# B&R Automation Studio project Panasonic_LinkaPowerCP2_A2021055 (part 29)

#### Main.st - Init, cyclic, exit code
```iecst
PROGRAM _INIT
	(* Insert code here *)

END_PROGRAM

PROGRAM _CYCLIC

		//Volanie funkcie SequenceControl//
	SequenceControl(SC:= SC_P3_LeakageTestB);

	//Volanie podprogramov//
	OvlCentrovacky;
	OvlHornehoPritlaku;
	IOLinkKomunikacia;
	COM_Tester;

	//Reset sekcie //
	IF P3_LeakageTestB.Reset THEN
		SC_P3_LeakageTestB.Step:= 0;
		P3_LeakageTestB.Reset:= FALSE;
	ELSIF NOT Safety.STAV.Linka_ZonaCS_AKTIVNA THEN
		SC_P3_LeakageTestB.Step:= 0;
	END_IF

	CASE SC_P3_LeakageTestB.Step OF

		0:
			SC_P3_LeakageTestB.StepName:='0 - Nulovanie';
			SC_OvlCentrovacky.Step:= 0;
			SC_OvlHornehoPritlaku.Step:= 0;
			P3_LeakageTestB.Automat:= FALSE;
			P3_LeakageTestB.KoniecCyklu:= FALSE;
			P3_LeakageTestB.Manual:= FALSE;
			P3_LeakageTestB.STAV.PoINIT:= FALSE;
			P3_LeakageTestB.OUT.ZasunStoper:= FALSE;
			P3_LeakageTestB.OUT.Kopito_VYSUN:= FALSE;
			P3_LeakageTestB.OUT.Kopito_ZASUN:= TRUE;
			P3_LeakageTestB.RFID_hlava.PrecitajChipRFID:= FALSE;
			P3_LeakageTestB.CMD.RR_TestovaciaSekvencia_START:= FALSE;
			P3_LeakageTestB.CMD.RR_VysunSpodneKopito:= FALSE;
			P3_LeakageTestB.CMD.RR_HornyPritlak_VYSUN:= FALSE;
			P3_LeakageTestB.CMD.RR_HornyPritlak_ZASUN:= FALSE;
			P3_LeakageTestB.STAV.RR_TestovaciaSekvencia_BUSY:= FALSE;
			TRCB_P3_LeakageTestB_ST8B.CMD.VyziadajStavPaletky_TYP1:= FALSE;
			TRCB_P3_LeakageTestB_ST8B.CMD.PriradQRkodFiltra_TYP3:= FALSE;
			TRCB_P3_LeakageTestB_ST8B.CMD.OdosliStavPaletky_TYP2:= FALSE;
			TRCB_P3_LeakageTestB_ST8B.CMD.VyziadajStavPanatrace_TYP4:= FALSE;
			AteqLeakageTester_B.CitajParametreTestera:= FALSE;
			AteqLeakageTester_B.START_Testovania:= FALSE;
			P34_Vizu.ZobrazHL2_ST8:= FALSE;
			P34_Vizu.ZobrazHL4_ST8:= FALSE;
			TRCB_P3_LeakTestB_OpatovnyDopyt:= FALSE;
			TRCB_P3_LeakTestB_PaletkaNG:= FALSE;
			PocetDopytovNaServer:= 0;
			PocetOpakovaniTestu:= 0;
			OpakovanyTest:= FALSE;
			TestovaciKus:= FALSE;
			P3_LeakageTestB_Taktime.IN.START_MeraniaCasu:= FALSE;
			P3_LeakageTestB_Taktime.IN.START_MeraniaStratovehoCasu:= FALSE;

			P3_ZdvizkaPredLeakTestB.STAV.PrebiehaVyvezeniePaletky:= FALSE;
			P3_LeakageTestB.STAV.PrebiehaVyvezeniePaletky:= FALSE;

			IF Safety.STAV.Linka_ZonaCS_AKTIVNA AND
				Safety.STAV.P3_ZonaBunky_AKTIVNA AND
				P3_Pracovisko.STAV.HardwareBunky_OK AND
				NOT P3_Pracovisko.STAV.Porucha_ST1 AND
				NOT P3_Pracovisko.STAV.Porucha_ST2 AND
				NOT P3_Pracovisko.STAV.Porucha_ST3 AND
				NOT P3_Pracovisko.STAV.Porucha_ST4 AND
				NOT P3_Pracovisko.STAV.Porucha_ST5 AND
				NOT P3_Pracovisko.STAV.Porucha_ST6 AND
				NOT P3_Pracovisko.STAV.Porucha_ST7 AND
				NOT P3_Pracovisko.STAV.Porucha_ST8 THEN
				SC_P3_LeakageTestB.ResetStep:= TRUE;
				SC_P3_LeakageTestB.Step:= 1;
			END_IF

		1:
			SC_P3_LeakageTestB.StepName:='1 - Cakam na spustenie vyroby';
			P3_LeakageTestB.KoniecCyklu:= FALSE;
			IF P3_LeakageTestB.Automat THEN
				SC_P3_LeakageTestB.Step:= 2;
			ELSIF P3_LeakageTestB.Manual THEN
				SC_P3_LeakageTestB.Step:= 700;
			END_IF

			//********************************************************Inicializácia****************************************************************************//

		2:
			SC_P3_LeakageTestB.StepName:='2 - Inicializacia - cakam na spustenie inicializacie';
			SC_P3_LeakageTestB.IdleTime.PT:= T#500ms;
			SC_P3_LeakageTestB.AlarmTime.PT:= T#5s;
			SC_P3_LeakageTestB.IdleTime.IN:= TRUE;

			IF SC_P3_LeakageTestB.IdleTime.Q THEN
				SC_P3_LeakageTestB.ResetStep:= TRUE;
				SC_P3_LeakageTestB.Step:= 5;
			END_IF

		5:
			SC_P3_LeakageTestB.StepName:='5 - Inicializacia - zasunutie horneho pritlaku';
			SC_P3_LeakageTestB.IdleTime.PT:= T#2s;
			SC_P3_LeakageTestB.AlarmTime.PT:= T#5s;

			IF NOT SC_P3_LeakageTestB.Switch1 THEN
				HornyPritlak_ZASUN:= TRUE;
				SC_P3_LeakageTestB.Switch1:= TRUE;
			END_IF

			IF P3_LeakageTestB.IN.HornyPritlak_ZASUNUTY THEN
				SC_P3_LeakageTestB.ResetStep:= TRUE;
				SC_P3_LeakageTestB.Step:= 8;
			END_IF

		8:
			SC_P3_LeakageTestB.StepName:='8 - Inicializacia - zasunutie centrovacky';
			SC_P3_LeakageTestB.IdleTime.PT:= T#4s;
			SC_P3_LeakageTestB.AlarmTime.PT:= T#5s;

			IF NOT SC_P3_LeakageTestB.Switch1 THEN
				Centrovacku_ZASUN:= TRUE;
				SC_P3_LeakageTestB.Switch1:= TRUE;
			END_IF

			IF P3_LeakageTestB.IN.Centrovanie_ZASUNUTE THEN
				SC_P3_LeakageTestB.ResetStep:= TRUE;
				SC_P3_LeakageTestB.Step:= 10;
			END_IF

		10:
			SC_P3_LeakageTestB.StepName:='10 - Inicializacia - kontrola typu zalozeneho kopita';
			SC_P3_LeakageTestB.IdleTime.PT:= T#4s;
			SC_P3_LeakageTestB.AlarmTime.PT:= T#5s;

			IF Linka.PAR.ZvolenyModel = '4F' AND P3_LeakageTestB.IN.PritomnostKopita AND P3_LeakageTestB.IN.Tester_TypKonektoru_4F THEN
				SC_P3_LeakageTestB.ResetStep:= TRUE;
				SC_P3_LeakageTestB.Step:= 13;
			ELSIF Linka.PAR.ZvolenyModel = '5F' AND P3_LeakageTestB.IN.PritomnostKopita AND P3_LeakageTestB.IN.Tester_TypKonektoru_5F_5H THEN
				SC_P3_LeakageTestB.ResetStep:= TRUE;
				SC_P3_LeakageTestB.Step:= 13;
			ELSIF Linka.PAR.ZvolenyModel = '5H' AND P3_LeakageTestB.IN.PritomnostKopita AND P3_LeakageTestB.IN.Tester_TypKonektoru_5F_5H THEN
				SC_P3_LeakageTestB.ResetStep:= TRUE;
				SC_P3_LeakageTestB.Step:= 13;
			ELSE
				P34_Alarmy[315]:= TRUE;
				P3_Pracovisko.STAV.Porucha_ST6:= TRUE;
			END_IF

		13:
			SC_P3_LeakageTestB.StepName:='13 - Inicializacia - hladanie paletky';
			SC_P3_LeakageTestB.IdleTime.PT:= T#5s;
			SC_P3_LeakageTestB.AlarmTime.PT:= T#5s;

			SC_P3_LeakageTestB.IdleTime.IN:= P3_Dopravniky.STAV.PoINIT;

			IF P3_LeakageTestB.CMD.RR_TestovaciaSekvencia_START THEN
				SC_P3_LeakageTestB.ResetStep:= TRUE;
				SC_P3_LeakageTestB.Step:= 120;
			ELSIF P3_LeakageTestB.RFID_hlava.PritomnostPaletky THEN
				SC_P3_LeakageTestB.ResetStep:= TRUE;
				SC_P3_LeakageTestB.Step:= 20;
			ELSIF SC_P3_LeakageTestB.IdleTime.Q THEN
				P3_LeakageTestB.STAV.PoINIT:= TRUE;
				SC_P3_LeakageTestB.ResetStep:= TRUE;
				SC_P3_LeakageTestB.Step:= 100;
			END_IF

		20:
			SC_P3_LeakageTestB.StepName:='20 - Inicializacia - precitanie cisla paletky';
			SC_P3_LeakageTestB.IdleTime.PT:= T#200ms;
			SC_P3_LeakageTestB.AlarmTime.PT:= T#5s;

			SC_P3_LeakageTestB.IdleTime.IN:= P3_LeakageTestB.RFID_hlava.PritomnostPaletky;

			IF SC_P3_LeakageTestB.IdleTime.Q AND NOT SC_P3_LeakageTestB.Switch1 THEN
				P3_LeakageTestB.RFID_hlava.PrecitajChipRFID:= TRUE;
				i:= 0;
				SC_P3_LeakageTestB.Switch1:= TRUE;
			END_IF

			IF P3_LeakageTestB.RFID_hlava.Stav_CitanieZapis_OK AND P3_LeakageTestB.RFID_hlava.PrecitaneCisloPaletky <> 0 THEN
				i:= P3_LeakageTestB.RFID_hlava.PrecitaneCisloPaletky;
				P3_LeakageTestB.PAR.CisloPaletky:= P3_LeakageTestB.RFID_hlava.PrecitaneCisloPaletky;
				P3_LeakageTestB.RFID_hlava.PrecitajChipRFID:= FALSE;
				SC_P3_LeakageTestB.ResetStep:= TRUE;
				SC_P3_LeakageTestB.Step:= 23;
			END_IF

		23:
			SC_P3_LeakageTestB.StepName:='23 - Inicializacia - priradenie indexu paletky na zaklade precitanej hodnoty';
			SC_P3_LeakageTestB.IdleTime.PT:= T#200ms;
			SC_P3_LeakageTestB.AlarmTime.PT:= T#5s;

			IF i<> 0 THEN
				P3_LeakageTestB.PAR.CisloPaletky_STRING:= USINT_TO_STRING(i);
				Paletka[i].PAR.CisloPaletky:= USINT_TO_STRING(i);
				SC_P3_LeakageTestB.ResetStep:= TRUE;
				SC_P3_LeakageTestB.Step:= 30;
			ELSE
				P34_Alarmy[312]:= TRUE;
				P3_Pracovisko.STAV.Porucha_ST6:= TRUE;
			END_IF

		30:
			SC_P3_LeakageTestB.StepName:='30 - Inicializacia - kontrola stavu paletky';
			SC_P3_LeakageTestB.IdleTime.PT:= T#200ms;
			SC_P3_LeakageTestB.AlarmTime.PT:= T#5s;

			IF Paletka[i].STAV.StavPaletky = '' THEN
				Paletka[i].STAV.StavPaletky:= 'NG';
				SC_P3_LeakageTestB.ResetStep:= TRUE;
				SC_P3_LeakageTestB.Step:= 560;
			ELSIF Paletka[i].STAV.StavPaletky = 'PRECH' THEN
				P3_LeakageTestB.STAV.PoINIT:= TRUE;
				SC_P3_LeakageTestB.ResetStep:= TRUE;
				SC_P3_LeakageTestB.Step:= 560;
			ELSIF Paletka[i].STAV.StavPaletky = 'TEST' AND Paletka[i].STAV.CisloTestovacejStanice = 'ST_8A,8B' THEN
				IF P3_LeakageTestB.STAV.Tester_ON THEN
					TestovaciKus:= TRUE;
					P3_LeakageTestB.STAV.PoINIT:= TRUE;
					SC_P3_LeakageTestB.ResetStep:= TRUE;
					SC_P3_LeakageTestB.Step:= 110;
				ELSE
					P3_LeakageTestB.STAV.PoINIT:= TRUE;
					SC_P3_LeakageTestB.ResetStep:= TRUE;
					SC_P3_LeakageTestB.Step:= 560;
				END_IF
			ELSIF Paletka[i].STAV.StavPaletky = 'TEST' AND Paletka[i].STAV.CisloTestovacejStanice <> 'ST_8A,8B' THEN
				P3_LeakageTestB.STAV.PoINIT:= TRUE;
				SC_P3_LeakageTestB.ResetStep:= TRUE;
				SC_P3_LeakageTestB.Step:= 560;
			ELSIF Paletka[i].STAV.StavPaletky = 'REV' AND Paletka[i].STAV.CisloRevorkovejStanice = 'ST_8A,8B' THEN
				IF P3_LeakageTestB.STAV.Tester_ON THEN
					Paletka[i].STAV.StavPaletky:= 'OK';
					P3_LeakageTestB.STAV.PoINIT:= TRUE;
					SC_P3_LeakageTestB.ResetStep:= TRUE;
					SC_P3_LeakageTestB.Step:= 110;
				ELSE
					P3_LeakageTestB.STAV.PoINIT:= TRUE;
					SC_P3_LeakageTestB.ResetStep:= TRUE;
					SC_P3_LeakageTestB.Step:= 560;
				END_IF
			ELSIF Paletka[i].STAV.StavPaletky = 'REV' AND Paletka[i].STAV.CisloRevorkovejStanice <> 'ST_8A,8B' THEN
				P3_LeakageTestB.STAV.PoINIT:= TRUE;
				SC_P3_LeakageTestB.ResetStep:= TRUE;
				SC_P3_LeakageTestB.Step:= 560;
			ELSIF Paletka[i].STAV.StavPaletky = 'OK' THEN
				IF P3_LeakageTestB.STAV.Tester_ON THEN
					SC_P3_LeakageTestB.ResetStep:= TRUE;
					SC_P3_LeakageTestB.Step:= 33;
				ELSE
					P3_LeakageTestB.STAV.PoINIT:= TRUE;
					SC_P3_LeakageTestB.ResetStep:= TRUE;
					SC_P3_LeakageTestB.Step:= 560;
				END_IF
			ELSIF Paletka[i].STAV.StavPaletky = 'NG' THEN
				P3_LeakageTestB.STAV.PoINIT:= TRUE;
				SC_P3_LeakageTestB.ResetStep:= TRUE;
				SC_P3_LeakageTestB.Step:= 560;
			END_IF

		33:
			SC_P3_LeakageTestB.StepName:='33 - Inicializacia - kontrola uzavretia komunikacie';
			SC_P3_LeakageTestB.IdleTime.PT:= T#200ms;
			SC_P3_LeakageTestB.AlarmTime.PT:= T#5s;

			IF Paletka[i].STAV.Komunikacia_DONE THEN
				P3_LeakageTestB.STAV.PoINIT:= TRUE;
				SC_P3_LeakageTestB.ResetStep:= TRUE;
				SC_P3_LeakageTestB.Step:= 560;
			ELSE
				P3_LeakageTestB.STAV.PoINIT:= TRUE;
				SC_P3_LeakageTestB.ResetStep:= TRUE;
				SC_P3_LeakageTestB.Step:= 100;
			END_IF

			//********************************************************Automatický režim****************************************************************************//

		100:
			SC_P3_LeakageTestB.StepName:='100 - Automaticky Rezim - cakam na príchod paletky na stoper';
			SC_P3_LeakageTestB.IdleTime.PT:= T#200ms;
			SC_P3_LeakageTestB.AlarmTime.PT:= T#5s;

			SC_P3_LeakageTestB.IdleTime.IN:= P3_LeakageTestB.RFID_hlava.PritomnostPaletky;

			IF P3_LeakageTestB.RFID_hlava.PritomnostPaletky THEN
				P3_ZdvizkaPredLeakTestB.STAV.PrebiehaVyvezeniePaletky:= FALSE;
			END_IF

			IF NOT SC_P3_LeakageTestB.Switch1 AND P3_LeakageTestB.RFID_hlava.PritomnostPaletky THEN
				P3_LeakageTestB_Taktime.IN.START_MeraniaCasu:= TRUE;
				P3_LeakageTestB_Taktime.IN.ZAPIS_MeraniaCasu:= TRUE;
				P3_LeakageTestB_Taktime.IN.ZAPIS_StratovyCas:= TRUE;
				Buffer_10.Hodnota:= P3_LeakageTestB_Taktime.OUT.StratoveSekundy;
				Buffer_10.ZapisHodnotu:= TRUE;
				SC_P3_LeakageTestB.Switch1:= TRUE;
			END_IF

			IF P3_LeakageTestB.KoniecCyklu THEN
				SC_P3_LeakageTestB.ResetStep:= TRUE;
				SC_P3_LeakageTestB.Step:= 0;
			ELSIF SC_P3_LeakageTestB.IdleTime.Q THEN
				SC_P3_LeakageTestB.ResetStep:= TRUE;
				SC_P3_LeakageTestB.Step:= 101;
			END_IF

		101:
			SC_P3_LeakageTestB.StepName:='101 - Automaticky Rezim - precitanie cisla paletky';
			SC_P3_LeakageTestB.IdleTime.PT:= T#200ms;
			SC_P3_LeakageTestB.AlarmTime.PT:= T#5s;
			SC_P3_LeakageTestB.IdleTime.IN:= TRUE;

			IF NOT SC_P3_LeakageTestB.Switch1 THEN
				P3_LeakageTestB.RFID_hlava.PrecitajChipRFID:= TRUE;
				i:= 0;
				SC_P3_LeakageTestB.Switch1:= TRUE;
			END_IF

			IF P3_LeakageTestB.RFID_hlava.Stav_CitanieZapis_OK AND P3_LeakageTestB.RFID_hlava.PrecitaneCisloPaletky <> 0 THEN
				i:= P3_LeakageTestB.RFID_hlava.PrecitaneCisloPaletky;
				P3_LeakageTestB.PAR.CisloPaletky:= P3_LeakageTestB.RFID_hlava.PrecitaneCisloPaletky;
				P3_LeakageTestB.RFID_hlava.PrecitajChipRFID:= FALSE;
				SC_P3_LeakageTestB.ResetStep:= TRUE;
				SC_P3_LeakageTestB.Step:= 102;
			END_IF

		102:
			SC_P3_LeakageTestB.StepName:='102 - Automaticky Rezim - priradenie indexu paletky na zaklade precitanej hodnoty';
			SC_P3_LeakageTestB.IdleTime.PT:= T#200ms;
			SC_P3_LeakageTestB.AlarmTime.PT:= T#5s;

			IF i<> 0 THEN
				P3_LeakageTestB.PAR.CisloPaletky_STRING:= USINT_TO_STRING(i);
				Paletka[i].PAR.CisloPaletky:= USINT_TO_STRING(i);
				SC_P3_LeakageTestB.ResetStep:= TRUE;
				SC_P3_LeakageTestB.Step:= 103;
			ELSE
				P34_Alarmy[312]:= TRUE;
				P3_Pracovisko.STAV.Porucha_ST6:= TRUE;
			END_IF

		103:
			SC_P3_LeakageTestB.StepName:='103 - Automaticky Rezim - kontrola stavu paletky';
			SC_P3_LeakageTestB.IdleTime.PT:= T#200ms;
			SC_P3_LeakageTestB.AlarmTime.PT:= T#5s;

			IF Paletka[i].STAV.StavPaletky = '' THEN
				Paletka[i].STAV.StavPaletky:= 'NG';
				SC_P3_LeakageTestB.ResetStep:= TRUE;
				SC_P3_LeakageTestB.Step:= 560;
			ELSIF Paletka[i].STAV.StavPaletky = 'PRECH' THEN
				SC_P3_LeakageTestB.ResetStep:= TRUE;
				SC_P3_LeakageTestB.Step:= 560;
			ELSIF Paletka[i].STAV.StavPaletky = 'TEST' AND Paletka[i].STAV.CisloTestovacejStanice = 'ST_8A,8B' THEN
				IF P3_LeakageTestB.STAV.Tester_ON THEN
					TestovaciKus:= TRUE;
					SC_P3_LeakageTestB.ResetStep:= TRUE;
					SC_P3_LeakageTestB.Step:= 110;
				ELSE
					SC_P3_LeakageTestB.ResetStep:= TRUE;
					SC_P3_LeakageTestB.Step:= 560;
				END_IF
			ELSIF Paletka[i].STAV.StavPaletky = 'TEST' AND Paletka[i].STAV.CisloTestovacejStanice <> 'ST_8A,8B' THEN
				SC_P3_LeakageTestB.ResetStep:= TRUE;
				SC_P3_LeakageTestB.Step:= 560;
			ELSIF Paletka[i].STAV.StavPaletky = 'REV' AND Paletka[i].STAV.CisloRevorkovejStanice = 'ST_8A,8B' THEN
				IF P3_LeakageTestB.STAV.Tester_ON THEN
					Paletka[i].STAV.StavPaletky:= 'OK';
					SC_P3_LeakageTestB.ResetStep:= TRUE;
					SC_P3_LeakageTestB.Step:= 110;
				ELSE
					SC_P3_LeakageTestB.ResetStep:= TRUE;
					SC_P3_LeakageTestB.Step:= 560;
				END_IF
			ELSIF Paletka[i].STAV.StavPaletky = 'REV' AND Paletka[i].STAV.CisloRevorkovejStanice <> 'ST_8A,8B' THEN
				SC_P3_LeakageTestB.ResetStep:= TRUE;
				SC_P3_LeakageTestB.Step:= 560;
			ELSIF Paletka[i].STAV.StavPaletky = 'OK' THEN
				IF P3_LeakageTestB.STAV.Tester_ON THEN
					SC_P3_LeakageTestB.ResetStep:= TRUE;
					SC_P3_LeakageTestB.Step:= 110;
				ELSE
					SC_P3_LeakageTestB.ResetStep:= TRUE;
					SC_P3_LeakageTestB.Step:= 560;
				END_IF
			ELSIF Paletka[i].STAV.StavPaletky = 'NG' THEN
				SC_P3_LeakageTestB.ResetStep:= TRUE;
				SC_P3_LeakageTestB.Step:= 560;
			END_IF

		110:
			SC_P3_LeakageTestB.StepName:='110 - Automaticky Rezim - vyziadanie stavu komunikacie zo serverom';
			SC_P3_LeakageTestB.IdleTime.PT:= T#200ms;
			SC_P3_LeakageTestB.AlarmTime.PT:= T#10s;

			IF Linka.KOM_Panatrace_OFF THEN
				SC_P3_LeakageTestB.ResetStep:= TRUE;
				SC_P3_LeakageTestB.Step:= 120;
			ELSIF NOT SC_P3_LeakageTestB.Switch1 THEN
				TRCB_P3_LeakageTestB_ST8B.CMD.VyziadajStavPanatrace_TYP4:= TRUE;
				Centrovacku_VYSUN:= TRUE;
				P3_LeakageTestB_Taktime.IN.START_MeraniaStratovehoCasu:= TRUE;
				SC_P3_LeakageTestB.Switch1:= TRUE;
			END_IF

			IF TRCB_P3_LeakageTestB_ST8B.STATUS.KomunikaciaUkoncena THEN
				TRCB_P3_LeakageTestB_ST8B.CMD.VyziadajStavPanatrace_TYP4:= FALSE;
				P3_LeakageTestB_Taktime.IN.START_MeraniaStratovehoCasu:= FALSE;
				SC_P3_LeakageTestB.ResetStep:= TRUE;
				SC_P3_LeakageTestB.Step:= 111;
			ELSIF TRCB_P3_LeakageTestB_ST8B.STATUS.KomunikaciaError THEN
				TRCB_P3_LeakageTestB_ST8B.CMD.VyziadajStavPanatrace_TYP4:= FALSE;
				P3_LeakageTestB_Taktime.IN.START_MeraniaStratovehoCasu:= FALSE;
				SC_P3_LeakageTestB.ResetStep:= TRUE;
				SC_P3_LeakageTestB.Step:= 112;
			END_IF

		111:
			SC_P3_LeakageTestB.StepName:='111 - Automaticky Rezim - kontrola odpovede servera';
			SC_P3_LeakageTestB.IdleTime.PT:= T#200ms;
			SC_P3_LeakageTestB.AlarmTime.PT:= T#5s;

			IF NOT TRCB_P3_LeakageTestB_ST8B.STATUS.KomunikaciaUkoncena THEN
				IF TRCB_P3_LeakageTestB_ST8B.OUTPUTS.DruhCinnostiNaPaletke = '0;Generating' THEN
					SC_P3_LeakageTestB.ResetStep:= TRUE;
					SC_P3_LeakageTestB.Step:= 112;
				ELSIF TRCB_P3_LeakageTestB_ST8B.OUTPUTS.DruhCinnostiNaPaletke = '1;Request' THEN
					SC_P3_LeakageTestB.ResetStep:= TRUE;
					SC_P3_LeakageTestB.Step:= 115;
				ELSIF TRCB_P3_LeakageTestB_ST8B.OUTPUTS.DruhCinnostiNaPaletke = '2;Report' THEN
					SC_P3_LeakageTestB.ResetStep:= TRUE;
					SC_P3_LeakageTestB.Step:= 120;
				ELSIF TRCB_P3_LeakageTestB_ST8B.OUTPUTS.DruhCinnostiNaPaletke = '3;Wedding' THEN
					SC_P3_LeakageTestB.ResetStep:= TRUE;
					SC_P3_LeakageTestB.Step:= 112;
				ELSIF TRCB_P3_LeakageTestB_ST8B.OUTPUTS.DruhCinnostiNaPaletke = '4;Status' THEN
					SC_P3_LeakageTestB.ResetStep:= TRUE;
					SC_P3_LeakageTestB.Step:= 112;
				ELSIF TRCB_P3_LeakageTestB_ST8B.OUTPUTS.DruhCinnostiNaPaletke = '5;' THEN
					SC_P3_LeakageTestB.ResetStep:= TRUE;
					SC_P3_LeakageTestB.Step:= 112;
				ELSE
					SC_P3_LeakageTestB.ResetStep:= TRUE;
					SC_P3_LeakageTestB.Step:= 112;
				END_IF
			END_IF

		112:
			SC_P3_LeakageTestB.StepName:='112 - Automaticky Rezim - rozhodnutie obsluhy po chybe komunikacie s Panatrace';
			SC_P3_LeakageTestB.IdleTime.PT:= T#200ms;
			SC_P3_LeakageTestB.AlarmTime.PT:= T#5s;

			P34_Vizu.ZobrazHL4_ST8:= TRUE;

			IF TRCB_P3_LeakTestB_OpatovnyDopyt THEN
				TRCB_P3_LeakTestB_OpatovnyDopyt:= FALSE;
				P34_Vizu.ZobrazHL4_ST8:= FALSE;
				SC_P3_LeakageTestB.ResetStep:= TRUE;
				SC_P3_LeakageTestB.Step:= 110;
			ELSIF TRCB_P3_LeakTestB_PaletkaNG THEN
				TRCB_P3_LeakTestB_PaletkaNG:= FALSE;
				P34_Vizu.ZobrazHL4_ST8:= FALSE;
				Paletka[i].STAV.StavPaletky := 'NG';
				SC_P3_LeakageTestB.ResetStep:= TRUE;
				SC_P3_LeakageTestB.Step:= 118;
			END_IF

		115:
			SC_P3_LeakageTestB.StepName:='115 - Automaticky Rezim - vyziadanie stavu paletky zo servera, zacentrovanie paletky';
			SC_P3_LeakageTestB.IdleTime.PT:= T#200ms;
			SC_P3_LeakageTestB.AlarmTime.PT:= T#5s;
			SC_P3_LeakageTestB.IdleTime.IN:= TRUE;

			IF NOT SC_P3_LeakageTestB.Switch1 AND TRCB_P3_LeakageTestB_ST8B.STATUS.KOM_READY THEN
				TRCB_P3_LeakageTestB_ST8B.CMD.VyziadajStavPaletky_TYP1:= TRUE;
				P3_LeakageTestB_Taktime.IN.START_MeraniaStratovehoCasu:= TRUE;
				SC_P3_LeakageTestB.Switch1:= TRUE;
			END_IF

			IF TRCB_P3_LeakageTestB_ST8B.STATUS.KomunikaciaUkoncena THEN
				TRCB_P3_LeakageTestB_ST8B.CMD.VyziadajStavPaletky_TYP1:= FALSE;
				P3_LeakageTestB_Taktime.IN.START_MeraniaStratovehoCasu:= FALSE;
				SC_P3_LeakageTestB.ResetStep:= TRUE;
				SC_P3_LeakageTestB.Step:= 116;
			ELSIF TRCB_P3_LeakageTestB_ST8B.STATUS.KomunikaciaError THEN
				TRCB_P3_LeakageTestB_ST8B.CMD.VyziadajStavPaletky_TYP1:= FALSE;
				P3_LeakageTestB_Taktime.IN.START_MeraniaStratovehoCasu:= FALSE;
				SC_P3_LeakageTestB.ResetStep:= TRUE;
				SC_P3_LeakageTestB.Step:= 112;
			END_IF

		116:
			SC_P3_LeakageTestB.StepName:='116 - Automaticky Rezim - kontrola odpovede servera';
			SC_P3_LeakageTestB.IdleTime.PT:= T#200ms;
			SC_P3_LeakageTestB.AlarmTime.PT:= T#5s;

			IF NOT TRCB_P3_LeakageTestB_ST8B.STATUS.KomunikaciaUkoncena AND P3_LeakageTestB.IN.Centrovanie_VYSUNUTE THEN
				IF TRCB_P3_LeakageTestB_ST8B.OUTPUTS.PovolenieCinnostiNaPaletke = 'OK' THEN
					IF TRCB_P3_LeakageTestB_ST8B.OUTPUTS.DruhCinnostiNaPaletke  = 'PRD;ST8B' THEN
						SC_P3_LeakageTestB.ResetStep:= TRUE;
						SC_P3_LeakageTestB.Step:= 120;
					ELSIF TRCB_P3_LeakageTestB_ST8B.OUTPUTS.DruhCinnostiNaPaletke  = 'SMP;ST8A,ST8B' THEN
						SC_P3_LeakageTestB.ResetStep:= TRUE;
						SC_P3_LeakageTestB.Step:= 120;
					ELSIF TRCB_P3_LeakageTestB_ST8B.OUTPUTS.DruhCinnostiNaPaletke  = 'PRD;ST8A,ST8B' THEN
						SC_P3_LeakageTestB.ResetStep:= TRUE;
						SC_P3_LeakageTestB.Step:= 120;
					END_IF
				ELSIF TRCB_P3_LeakageTestB_ST8B.OUTPUTS.PovolenieCinnostiNaPaletke = 'NG' THEN
					SC_P3_LeakageTestB.ResetStep:= TRUE;
					SC_P3_LeakageTestB.Step:= 117;
				END_IF
			END_IF

		117:
			SC_P3_LeakageTestB.StepName:='115 - Automaticky Rezim - rozhodnutie obsluhy po odpovedi panatrace NG';
			SC_P3_LeakageTestB.IdleTime.PT:= T#200ms;
			SC_P3_LeakageTestB.AlarmTime.PT:= T#5s;

			P34_Vizu.ZobrazHL2_ST8:= TRUE;

			IF TRCB_P3_LeakTestB_OpatovnyDopyt THEN
				TRCB_P3_LeakTestB_OpatovnyDopyt:= FALSE;
				P34_Vizu.ZobrazHL2_ST8:= FALSE;
				SC_P3_LeakageTestB.ResetStep:= TRUE;
				SC_P3_LeakageTestB.Step:= 110;
			ELSIF TRCB_P3_LeakTestB_PaletkaNG THEN
				TRCB_P3_LeakTestB_PaletkaNG:= FALSE;
				P34_Vizu.ZobrazHL2_ST8:= FALSE;
				Paletka[i].STAV.StavPaletky := 'NG';
				SC_P3_LeakageTestB.ResetStep:= TRUE;
				SC_P3_LeakageTestB.Step:= 118;
			END_IF

		118:
			SC_P3_LeakageTestB.StepName:='118 - Automaticky Rezim - odcentrovanie paletky po odpovedi servera NG';
			SC_P3_LeakageTestB.IdleTime.PT:= T#200ms;
			SC_P3_LeakageTestB.AlarmTime.PT:= T#5s;

			IF NOT SC_P3_LeakageTestB.Switch1 THEN
				Centrovacku_ZASUN:= TRUE;
				SC_P3_LeakageTestB.Switch1:= TRUE;
			END_IF

			IF P3_LeakageTestB.IN.Centrovanie_ZASUNUTE THEN
				SC_P3_LeakageTestB.ResetStep:= TRUE;
				SC_P3_LeakageTestB.Step:= 560;
			END_IF

			//Zatvorenie Leakage testera//

		120:
			SC_P3_LeakageTestB.StepName:='120 - Automaticky Rezim - zacentrovanie paletky ';
			SC_P3_LeakageTestB.IdleTime.PT:= T#200ms;
			SC_P3_LeakageTestB.AlarmTime.PT:= T#5s;

			IF NOT SC_P3_LeakageTestB.Switch1 THEN
				Centrovacku_VYSUN:= TRUE;
				SC_P3_LeakageTestB.Switch1:= TRUE;
			END_IF

			IF P3_LeakageTestB.IN.Centrovanie_VYSUNUTE THEN
				SC_P3_LeakageTestB.ResetStep:= TRUE;
				SC_P3_LeakageTestB.Step:= 123;
			END_IF

		123:
			SC_P3_LeakageTestB.StepName:='123 - Automaticky Rezim - vysunutie horneho pritlaku ';
			SC_P3_LeakageTestB.IdleTime.PT:= T#3s;
			SC_P3_LeakageTestB.AlarmTime.PT:= T#5s;

			IF NOT SC_P3_LeakageTestB.Switch1 THEN
				HornyPritlak_VYSUN:= TRUE;
				SC_P3_LeakageTestB.Switch1:= TRUE;
			END_IF

			IF P3_LeakageTestB.IN.HornyPritlak_VYSUNUTY THEN
				SC_P3_LeakageTestB.ResetStep:= TRUE;
				SC_P3_LeakageTestB.Step:= 125;
			END_IF

		125:
			SC_P3_LeakageTestB.StepName:='125 - Automaticky Rezim - vysunutie spodneho kopita';
			SC_P3_LeakageTestB.IdleTime.PT:= T#1s;
			SC_P3_LeakageTestB.AlarmTime.PT:= T#5s;
			SC_P3_LeakageTestB.IdleTime.IN:= TRUE;

			IF P3_LeakageTestB.IN.PritomnostKopita AND P3_LeakageTestB.IN.Kopito_ZASUNUTE THEN
				P3_LeakageTestB.OUT.Kopito_ZASUN:= FALSE;
				P3_LeakageTestB.OUT.Kopito_VYSUN:= TRUE;
				SC_P3_LeakageTestB.ResetStep:= TRUE;
				SC_P3_LeakageTestB.Step:= 128;
			END_IF

		128:
			SC_P3_LeakageTestB.StepName:='128 - Automaticky Rezim - cakam na vysunutie kopita';
			SC_P3_LeakageTestB.IdleTime.PT:= T#200ms;
			SC_P3_LeakageTestB.AlarmTime.PT:= T#300ms;

			SC_P3_LeakageTestB.IdleTime.IN:= NOT P3_LeakageTestB.IN.Kopito_ZASUNUTE;

			IF SC_P3_LeakageTestB.IdleTime.Q THEN
				P3_LeakageTestB.OUT.PneuZamokCentrovania_ODOMKNI:= FALSE;
				P3_LeakageTestB.OUT.PneuZamokZvonu_ODOMKNI:= FALSE;
				SC_P3_LeakageTestB.ResetStep:= TRUE;
				SC_P3_LeakageTestB.Step:= 130;
			END_IF

		130:
			SC_P3_LeakageTestB.StepName:='130 - Automaticky Rezim - spustenie testera';
			SC_P3_LeakageTestB.IdleTime.PT:= T#4s800ms;
			SC_P3_LeakageTestB.AlarmTime.PT:= T#5s;

			IF NOT SC_P3_LeakageTestB.Switch1 AND AteqLeakageTester_B.Stav_READY THEN
				AteqLeakageTester_B.START_Testovania:= TRUE;
				SC_P3_LeakageTestB.IdleTime.IN:= TRUE;
				SC_P3_LeakageTestB.Switch1:= TRUE;
			END_IF

			IF NOT AteqLeakageTester_B.Stav_READY AND AteqLeakageTester_B.Stav_START_DONE AND NOT AteqLeakageTester_B.VysledokTestovania_OK AND NOT AteqLeakageTester_B.VysledokTestovania_NG AND SC_P3_LeakageTestB.IdleTime.Q THEN
				SC_P3_LeakageTestB.ResetStep:= TRUE;
				SC_P3_LeakageTestB.Step:= 133;
			END_IF

		133:
			SC_P3_LeakageTestB.StepName:='133 - Automaticky Rezim - nacitanie parametrov testera';
			SC_P3_LeakageTestB.IdleTime.PT:= T#500ms;
			SC_P3_LeakageTestB.AlarmTime.PT:= T#5s;

			IF AteqLeakageTester_B.Stav_READY THEN
				AteqLeakageTester_B.START_Testovania:= FALSE;
				AteqLeakageTester_B.CitajParametreTestera:= TRUE;
			END_IF

			SC_P3_LeakageTestB.IdleTime.IN:= AteqLeakageTester_B.Stav_CitanieParametrov_OK;

			IF AteqLeakageTester_B.Stav_CitanieParametrov_OK AND SC_P3_LeakageTestB.IdleTime.Q THEN
				Reports.LeakageTest.CasPlnenia.StanicaB:= REAL_TO_STRING(AteqLeakageTester_B.CasPnenia);
				Reports.LeakageTest.CasStabilizacie.StanicaB:= REAL_TO_STRING(AteqLeakageTester_B.CasStabilizacie);
				Reports.LeakageTest.TlakPlnenia.StanicaB:= REAL_TO_STRING(AteqLeakageTester_B.TlakPlnenia);
				Reports.LeakageTest.ToleranciaPritlaku_MIN.StanicaB:= '';
				Reports.LeakageTest.ToleranciaPritlaku_MAX.StanicaB:= '';
				Reports.LeakageTest.TlakPritlaku.StanicaB:= REAL_TO_STRING(P3_LeakageTestB.PAR.PreratanyVyrovnavaciTlak_Bar);
				Reports.LeakageTest.TlakUniku.StanicaB:= REAL_TO_STRING(AteqLeakageTester_B.TlakUniku);
				Reports.LeakageTest.ToleranciaTlakUniku_MIN.StanicaB:= REAL_TO_STRING(AteqLeakageTester_B.Tolerancia * -1);
				Reports.LeakageTest.ToleranciaTlakUniku_MAX.StanicaB:= REAL_TO_STRING(AteqLeakageTester_B.Tolerancia);
				Reports.LeakageTest.Tolerancia.StanicaB:= REAL_TO_STRING(AteqLeakageTester_B.Tolerancia);
				AteqLeakageTester_B.CitajParametreTestera:= FALSE;
				IF P3_LeakageTestB.STAV.RR_TestovaciaSekvencia_BUSY THEN
					SC_P3_LeakageTestB.ResetStep:= TRUE;
					SC_P3_LeakageTestB.Step:= 150;
				ELSE
					SC_P3_LeakageTestB.ResetStep:= TRUE;
					SC_P3_LeakageTestB.Step:= 135;
				END_IF
			END_IF

		135:
			SC_P3_LeakageTestB.StepName:='135 - Automaticky Rezim - kontrola výsledku testu';
			SC_P3_LeakageTestB.IdleTime.PT:= T#1s;
			SC_P3_LeakageTestB.AlarmTime.PT:= T#5s;

			IF AteqLeakageTester_B.VysledokTestovania_OK THEN
				Paletka[i].STAV.LeakageTest_Ukonceny:= TRUE;
				Reports.LeakageTest.VyslednyReport.StanicaB:= 'PASS';
				Paletka[i].PAR.StavPowerCP:= 'PASS';
				IF Paletka[i].STAV.StavPaletky <> 'TEST'THEN
					Paletka[i].STAV.StavPaletky:= 'OK';
				END_IF
				PocetOpakovaniTestu:= 0;
				OpakovanyTest:= FALSE;
				SC_P3_LeakageTestB.ResetStep:= TRUE;
				SC_P3_LeakageTestB.Step:= 150;
			ELSE
				IF NOT TestovaciKus THEN
					PocetOpakovaniTestu:= PocetOpakovaniTestu + 1;
					OpakovanyTest:= TRUE;
				END_IF
				Reports.LeakageTest.VyslednyReport.StanicaB:= 'FAIL';
				Paletka[i].PAR.StavPowerCP:= 'FAIL';
				IF Paletka[i].STAV.StavPaletky <> 'TEST'THEN
					Paletka[i].STAV.StavPaletky:= 'NG';
				END_IF
				SC_P3_LeakageTestB.ResetStep:= TRUE;
				SC_P3_LeakageTestB.Step:= 150;
			END_IF

			//Otvorenie Leakage testera//

		150:
			SC_P3_LeakageTestB.StepName:='150 - Automaticky Rezim - zasunutie spodneho kopita ';
			SC_P3_LeakageTestB.IdleTime.PT:= T#200ms;
			SC_P3_LeakageTestB.AlarmTime.PT:= T#5s;

			P3_LeakageTestB.OUT.Kopito_VYSUN:= FALSE;
			P3_LeakageTestB.OUT.Kopito_ZASUN:= TRUE;

			IF P3_LeakageTestB.IN.Kopito_ZASUNUTE THEN
				SC_P3_LeakageTestB.ResetStep:= TRUE;
				SC_P3_LeakageTestB.Step:= 153;
			END_IF

		153:
			SC_P3_LeakageTestB.StepName:='153 - Automaticky Rezim - zasunutie horneho pritlaku';
			SC_P3_LeakageTestB.IdleTime.PT:= T#200ms;
			SC_P3_LeakageTestB.AlarmTime.PT:= T#5s;

			IF NOT SC_P3_LeakageTestB.Switch1 THEN
				HornyPritlak_ZASUN:= TRUE;
				Centrovacku_ZASUN:= TRUE;
				SC_P3_LeakageTestB.Switch1:= TRUE;
			END_IF

			IF P3_LeakageTestB.IN.HornyPritlak_ZASUNUTY THEN
				SC_P3_LeakageTestB.ResetStep:= TRUE;
				SC_P3_LeakageTestB.Step:= 155;
			END_IF

		155:
			SC_P3_LeakageTestB.StepName:='155 - Automaticky Rezim - odcentrovanie paletky ';
			SC_P3_LeakageTestB.IdleTime.PT:= T#200ms;
			SC_P3_LeakageTestB.AlarmTime.PT:= T#5s;

			IF NOT SC_P3_LeakageTestB.Switch1 THEN
				Centrovacku_ZASUN:= TRUE;
				SC_P3_LeakageTestB.Switch1:= TRUE;
			END_IF

			IF P3_LeakageTestB.IN.Centrovanie_ZASUNUTE THEN
				IF P3_LeakageTestB.STAV.RR_TestovaciaSekvencia_BUSY THEN
					P3_LeakageTestB.STAV.RR_TestovaciaSekvencia_BUSY:= FALSE;
					SC_P3_LeakageTestB.ResetStep:= TRUE;
					SC_P3_LeakageTestB.Step:= 700;
				ELSE
					SC_P3_LeakageTestB.ResetStep:= TRUE;
					SC_P3_LeakageTestB.Step:= 160;
				END_IF
			END_IF

		160:
			SC_P3_LeakageTestB.StepName:='160 - Automaticky Rezim - rozhodnutie o opakovani testu ';
			SC_P3_LeakageTestB.IdleTime.PT:= T#1s;
			SC_P3_LeakageTestB.AlarmTime.PT:= T#5s;
			SC_P3_LeakageTestB.IdleTime.IN:= TRUE;

			IF OpakovanyTest AND PocetOpakovaniTestu < 2 AND SC_P3_LeakageTestB.IdleTime.Q THEN
				SC_P3_LeakageTestB.ResetStep:= TRUE;
				SC_P3_LeakageTestB.Step:= 120;
			ELSIF OpakovanyTest AND PocetOpakovaniTestu >= 2 THEN
				PocetOpakovaniTestu:= 0;
				OpakovanyTest:= FALSE;
				SC_P3_LeakageTestB.ResetStep:= TRUE;
				SC_P3_LeakageTestB.Step:= 550;
			ELSIF NOT OpakovanyTest THEN
				PocetOpakovaniTestu:= 0;
				OpakovanyTest:= FALSE;
				SC_P3_LeakageTestB.ResetStep:= TRUE;
				SC_P3_LeakageTestB.Step:= 550;
			END_IF

			//**************************Odoslanie dát na server************************************//
		550:
			SC_P3_LeakageTestB.StepName:='550 - Automaticky Rezim - odoslanie stavu paletky na server';
			SC_P3_LeakageTestB.IdleTime.PT:= T#200ms;
			SC_P3_LeakageTestB.AlarmTime.PT:= T#5s;

			IF Linka.KOM_Panatrace_OFF THEN
				SC_P3_LeakageTestB.ResetStep:= TRUE;
				SC_P3_LeakageTestB.Step:= 560;
			ELSIF NOT SC_P3_LeakageTestB.Switch1 AND TRCB_P3_LeakageTestB_ST8B.STATUS.KOM_READY THEN
				TRCB_P3_LeakageTestB_ST8B.CMD.OdosliStavPaletky_TYP2:= TRUE;
				P3_LeakageTestB_Taktime.IN.START_MeraniaStratovehoCasu:= TRUE;
				SC_P3_LeakageTestB.Switch1:= TRUE;
			END_IF

			IF TRCB_P3_LeakageTestB_ST8B.STATUS.KomunikaciaUkoncena THEN
				TRCB_P3_LeakageTestB_ST8B.CMD.OdosliStavPaletky_TYP2:= FALSE;
				P3_LeakageTestB_Taktime.IN.START_MeraniaStratovehoCasu:= FALSE;
				SC_P3_LeakageTestB.ResetStep:= TRUE;
				SC_P3_LeakageTestB.Step:= 552;
			ELSIF TRCB_P3_LeakageTestB_ST8B.STATUS.KomunikaciaError THEN
				TRCB_P3_LeakageTestB_ST8B.CMD.OdosliStavPaletky_TYP2:= FALSE;
				P3_LeakageTestB_Taktime.IN.START_MeraniaStratovehoCasu:= FALSE;
				SC_P3_LeakageTestB.ResetStep:= TRUE;
				SC_P3_LeakageTestB.Step:= 557;
			END_IF

		552:
			SC_P3_LeakageTestB.StepName:='552 - Automaticky Rezim - kontrola odpovede servera';
			SC_P3_LeakageTestB.IdleTime.PT:= T#200ms;
			SC_P3_LeakageTestB.AlarmTime.PT:= T#5s;

			IF NOT TRCB_P3_LeakageTestB_ST8B.STATUS.KomunikaciaUkoncena THEN
				IF TRCB_P3_LeakageTestB_ST8B.OUTPUTS.PovolenieCinnostiNaPaletke = 'OK' THEN
					Paletka[i].STAV.Komunikacia_DONE:= TRUE;
					SC_P3_LeakageTestB.ResetStep:= TRUE;
					SC_P3_LeakageTestB.Step:= 560;
				ELSIF TRCB_P3_LeakageTestB_ST8B.OUTPUTS.PovolenieCinnostiNaPaletke = 'NG' THEN
					IF Paletka[i].STAV.StavPaletky <> 'TEST'THEN
						Paletka[i].STAV.StavPaletky:= 'NG';
					END_IF
					SC_P3_LeakageTestB.ResetStep:= TRUE;
					SC_P3_LeakageTestB.Step:= 560;
				END_IF
			END_IF

		555:
			SC_P3_LeakageTestB.StepName:='555 - Automaticky Rezim - vyziadanie stavu komunikacie zo serverom';
			SC_P3_LeakageTestB.IdleTime.PT:= T#200ms;
			SC_P3_LeakageTestB.AlarmTime.PT:= T#10s;

			IF NOT SC_P3_LeakageTestB.Switch1 AND TRCB_P3_LeakageTestB_ST8B.STATUS.KOM_READY THEN
				TRCB_P3_LeakageTestB_ST8B.CMD.VyziadajStavPanatrace_TYP4:= TRUE;
				SC_P3_LeakageTestB.Switch1:= TRUE;
			END_IF

			IF TRCB_P3_LeakageTestB_ST8B.STATUS.KomunikaciaUkoncena THEN
				TRCB_P3_LeakageTestB_ST8B.CMD.VyziadajStavPanatrace_TYP4:= FALSE;
				SC_P3_LeakageTestB.ResetStep:= TRUE;
				SC_P3_LeakageTestB.Step:= 556;
			ELSIF TRCB_P3_LeakageTestB_ST8B.STATUS.KomunikaciaError THEN
				TRCB_P3_LeakageTestB_ST8B.CMD.VyziadajStavPanatrace_TYP4:= FALSE;
				SC_P3_LeakageTestB.ResetStep:= TRUE;
				SC_P3_LeakageTestB.Step:= 557;
			END_IF

		556:
			SC_P3_LeakageTestB.StepName:='556 - Automaticky Rezim - kontrola odpovede servera';
			SC_P3_LeakageTestB.IdleTime.PT:= T#200ms;
			SC_P3_LeakageTestB.AlarmTime.PT:= T#5s;

			IF NOT TRCB_P3_LeakageTestB_ST8B.STATUS.KomunikaciaUkoncena THEN
				IF TRCB_P3_LeakageTestB_ST8B.OUTPUTS.DruhCinnostiNaPaletke = '0;Generating' THEN
					SC_P3_LeakageTestB.ResetStep:= TRUE;
					SC_P3_LeakageTestB.Step:= 557;
				ELSIF TRCB_P3_LeakageTestB_ST8B.OUTPUTS.DruhCinnostiNaPaletke = '1;Request' THEN
					SC_P3_LeakageTestB.ResetStep:= TRUE;
					SC_P3_LeakageTestB.Step:= 557;
				ELSIF TRCB_P3_LeakageTestB_ST8B.OUTPUTS.DruhCinnostiNaPaletke = '2;Report' THEN
					SC_P3_LeakageTestB.ResetStep:= TRUE;
					SC_P3_LeakageTestB.Step:= 550;
				ELSIF TRCB_P3_LeakageTestB_ST8B.OUTPUTS.DruhCinnostiNaPaletke = '3;Wedding' THEN
					SC_P3_LeakageTestB.ResetStep:= TRUE;
					SC_P3_LeakageTestB.Step:= 557;
				ELSIF TRCB_P3_LeakageTestB_ST8B.OUTPUTS.DruhCinnostiNaPaletke = '4;Status' THEN
					SC_P3_LeakageTestB.ResetStep:= TRUE;
					SC_P3_LeakageTestB.Step:= 557;
				ELSIF TRCB_P3_LeakageTestB_ST8B.OUTPUTS.DruhCinnostiNaPaletke = '5;' THEN
					SC_P3_LeakageTestB.ResetStep:= TRUE;
					SC_P3_LeakageTestB.Step:= 557;
				ELSE
					SC_P3_LeakageTestB.ResetStep:= TRUE;
					SC_P3_LeakageTestB.Step:= 557;
				END_IF
			END_IF

		557:
			SC_P3_LeakageTestB.StepName:='557 - Automaticky Rezim - rozhodnutie obsluhy po chybe komunikacie s Panatrace';
			SC_P3_LeakageTestB.IdleTime.PT:= T#200ms;
			SC_P3_LeakageTestB.AlarmTime.PT:= T#5s;

			P34_Vizu.ZobrazHL4_ST8:= TRUE;

			IF TRCB_P3_LeakTestB_OpatovnyDopyt THEN
				TRCB_P3_LeakTestB_OpatovnyDopyt:= FALSE;
				P34_Vizu.ZobrazHL4_ST8:= FALSE;
				SC_P3_LeakageTestB.ResetStep:= TRUE;
				SC_P3_LeakageTestB.Step:= 555;
			ELSIF TRCB_P3_LeakTestB_PaletkaNG THEN
				TRCB_P3_LeakTestB_PaletkaNG:= FALSE;
				P34_Vizu.ZobrazHL4_ST8:= FALSE;
				Paletka[i].STAV.StavPaletky := 'NG';
				SC_P3_LeakageTestB.ResetStep:= TRUE;
				SC_P3_LeakageTestB.Step:= 560;
			END_IF

			//***************************Vyvezenie paletky**********************************************//

		560:
			SC_P3_LeakageTestB.StepName:='560 - Automaticky Rezim - cakam na vyvezenie na zdvizku za leakage testom B';
			SC_P3_LeakageTestB.IdleTime.PT:= T#200ms;
			SC_P3_LeakageTestB.AlarmTime.PT:= T#5s;

			IF P3_LeakageTestB.KoniecCyklu THEN
				SC_P3_LeakageTestB.ResetStep:= TRUE;
				SC_P3_LeakageTestB.Step:= 0;
			ELSIF P3_Pracovisko.STAV.Porucha_ST6 THEN
				SC_P3_LeakageTestB.ResetStep:= TRUE;
				SC_P3_LeakageTestB.Step:= 0;
			ELSIF NOT P3_ZdvizkaZaLeakTestB.IN.PritomnostPaletky AND
				SC_P3_ZdvizkaZaLeakTestB.Step = 100 AND
				NOT P3_LeakageTestB.STAV.PrebiehaVyvezeniePaletky AND
				NOT P3_ZdvizkaZaLeakTestA.STAV.PrebiehaVyvezeniePaletkyNaTratB AND
				P3_ZdvizkaZaLeakTestB.IN.Zdvizka_StrednaPoloha AND
				P3_ZdvizkaZaLeakTestA.STAV.PoINIT AND
				P3_ZdvizkaZaLeakTestB.STAV.PoINIT THEN
				P3_LeakageTestB.OUT.ZasunStoper:= TRUE;
				P3_LeakageTestB.STAV.PrebiehaVyvezeniePaletky:= TRUE;
				SC_P3_LeakageTestB.ResetStep:= TRUE;
				SC_P3_LeakageTestB.Step:= 561;
			END_IF

		561:
			SC_P3_LeakageTestB.StepName:='561 - Automaticky Rezim - ukoncenie vyvazania na zdvizku za leakage testom B';
			SC_P3_LeakageTestB.IdleTime.PT:= T#200ms;
			SC_P3_LeakageTestB.AlarmTime.PT:= T#10s;

			SC_P3_LeakageTestB.IdleTime.IN:= NOT P3_LeakageTestB.RFID_hlava.PritomnostPaletky;
			SC_P3_LeakageTestB.AlarmTime.IN:= P3_LeakageTestB.RFID_hlava.PritomnostPaletky;

			IF NOT P3_LeakageTestB.RFID_hlava.PritomnostPaletky THEN
				P3_LeakageTestB.OUT.ZasunStoper:= FALSE;
				TestovaciKus:= FALSE;
				OpakovanyTest:= FALSE;
				PocetOpakovaniTestu:= 0;
				Paletka[i].PAR.StavPowerCP:= '';
				Paletka[i].STAV.Komunikacia_DONE:= FALSE;
				Reports.LeakageTest.CasPlnenia.StanicaB:= '';
				Reports.LeakageTest.VyslednyReport.StanicaB:= '';
				Reports.LeakageTest.CasStabilizacie.StanicaB:= '';
				Reports.LeakageTest.TlakPlnenia.StanicaB:= '';
				Reports.LeakageTest.ToleranciaPritlaku_MIN.StanicaB:= '';
				Reports.LeakageTest.ToleranciaPritlaku_MAX.StanicaB:= '';
				Reports.LeakageTest.TlakPritlaku.StanicaB:= '';
				Reports.LeakageTest.TlakUniku.StanicaB:= '';
				Reports.LeakageTest.Tolerancia.StanicaB:= '';
				SC_P3_LeakageTestB.ResetStep:= TRUE;
				SC_P3_LeakageTestB.Step:= 100;
			ELSIF SC_P3_LeakageTestB.AlarmTime.Q THEN
				P34_Alarmy[358]:= TRUE;
				P3_Pracovisko.STAV.Porucha_ST6:= TRUE;
			END_IF

			//*******************************************************Manuálny režim*******************************************************************************//
		700:
			SC_P3_LeakageTestB.StepName:='700 - Manualny Rezim';
			SC_P3_LeakageTestB.IdleTime.PT:= T#8s;
			SC_P3_LeakageTestB.AlarmTime.PT:= T#5s;

			//Vysunutie spodneho kopita//
			IF P3_LeakageTestB.CMD.RR_VysunSpodneKopito THEN
				P3_LeakageTestB.OUT.Kopito_ZASUN:= FALSE;
				P3_LeakageTestB.OUT.Kopito_VYSUN:= TRUE;
			ELSE
				P3_LeakageTestB.OUT.Kopito_VYSUN:= FALSE;
				P3_LeakageTestB.OUT.Kopito_ZASUN:= TRUE;
			END_IF

			//Testovacia sekvencia//
			IF P3_LeakageTestB.CMD.RR_TestovaciaSekvencia_START THEN
				IF P3_LeakageTestB.RFID_hlava.PritomnostPaletky THEN
					P3_LeakageTestB.STAV.RR_TestovaciaSekvencia_BUSY:= TRUE;
					SC_P3_LeakageTestB.ResetStep:= TRUE;
					SC_P3_LeakageTestB.Step:= 120;
				END_IF
				P3_LeakageTestB.CMD.RR_TestovaciaSekvencia_START:= FALSE;
			END_IF

			//Ovládanie centrovania paletky//
			IF P3_LeakageTestB.CMD.RR_VysunCentrovanie THEN
				P3_LeakageTestB.OUT.PneuZamokCentrovania_ODOMKNI:= TRUE;
				P3_LeakageTestB.OUT.Centrovanie_VYSUN:= TRUE;
			ELSE
				P3_LeakageTestB.OUT.PneuZamokCentrovania_ODOMKNI:= TRUE;
				P3_LeakageTestB.OUT.Centrovanie_VYSUN:= FALSE;
			END_IF

			//Ovládanie horného prítlaku//
			IF P3_LeakageTestB.CMD.RR_HornyPritlak_VYSUN THEN
				P3_LeakageTestB.OUT.PneuZamokZvonu_ODOMKNI:= TRUE;
				P3_LeakageTestB.OUT.HornyPritlak_ZASUN:= FALSE;
				P3_LeakageTestB.OUT.HornyPritlak_VYSUN:= TRUE;
				P3_LeakageTestB.CMD.RR_HornyPritlak_VYSUN:= FALSE;
			ELSIF P3_LeakageTestB.CMD.RR_HornyPritlak_ZASUN THEN
				P3_LeakageTestB.OUT.PneuZamokZvonu_ODOMKNI:= TRUE;
				P3_LeakageTestB.OUT.HornyPritlak_ZASUN:= TRUE;
				P3_LeakageTestB.OUT.HornyPritlak_VYSUN:= FALSE;
				P3_LeakageTestB.CMD.RR_HornyPritlak_ZASUN:= FALSE;
			END_IF

	END_CASE

END_PROGRAM

PROGRAM _EXIT
	(* Insert code here *)

END_PROGRAM
```

#### Variables.var - Local variables
```iecst
VAR
	SC_OvlCentrovacky : SequenceControlTyp;
	Centrovacku_VYSUN : BOOL;
	Centrovacku_ZASUN : BOOL;
	i : USINT;
	SC_OvlHornehoPritlaku : SequenceControlTyp := (0);
	HornyPritlak_VYSUN : BOOL := FALSE;
	HornyPritlak_ZASUN : BOOL := FALSE;
	CasPneniaREAL : REAL;
	CasStabilizacieREAL : REAL;
	TlakPlneniaREAL : REAL;
	ToleranciaREAL : REAL;
	TlakUnikuREAL : REAL;
	PocetDopytovNaServer : USINT := 0;
	PocetOpakovaniTestu : USINT := 0;
	TestovaciKus : BOOL := 0;
	OpakovanyTest : BOOL := 0;
	Triger_0 : BOOL := 0;
END_VAR
```

#### IOLinkKomunikacia.st
```iecst
ACTION IOLinkKomunikacia:

	//RFID snímač paletky//
	P3_LeakageTestB.RFID_hlava();

END_ACTION
```

#### OvlCentrovacky.st
```iecst
ACTION OvlCentrovacky:

	//Volanie funkcie SequenceControl//
	SequenceControl(SC:= SC_OvlCentrovacky);

	CASE SC_OvlCentrovacky.Step OF

		0:
			SC_OvlCentrovacky.StepName:= '0 - Nulovanie';
			Centrovacku_VYSUN:= FALSE;
			Centrovacku_ZASUN:= FALSE;

			IF SC_P3_LeakageTestB.Step <> 0 THEN
				SC_OvlCentrovacky.ResetStep:= TRUE;
				SC_OvlCentrovacky.Step:= 1;
			END_IF

		1:
			SC_OvlCentrovacky.StepName:= '1 - Rozhodnutie o cinnosti';
			IF Centrovacku_VYSUN THEN
				SC_OvlCentrovacky.Step:= 10;
			ELSIF Centrovacku_ZASUN THEN
				SC_OvlCentrovacky.Step:= 20;
			END_IF

		10:
			SC_OvlCentrovacky.StepName:= '10 - Vysunutie centrovacky';
			SC_OvlCentrovacky.IdleTime.PT:= T#3s;
			SC_OvlCentrovacky.AlarmTime.PT:= T#10s;

			IF P3_LeakageTestB.Automat THEN
				SC_OvlCentrovacky.AlarmTime.IN:= TRUE;
			ELSE
				SC_OvlCentrovacky.IdleTime.IN:= TRUE;
			END_IF

			IF NOT SC_OvlCentrovacky.Switch1 THEN
				P3_LeakageTestB.OUT.PneuZamokCentrovania_ODOMKNI:= TRUE;
                P3_LeakageTestB.OUT.Centrovanie_VYSUN:= TRUE;
				SC_OvlCentrovacky.Switch1:= TRUE;
			END_IF

			IF P3_LeakageTestB.IN.Centrovanie_VYSUNUTE OR SC_OvlCentrovacky.IdleTime.Q THEN
				SC_OvlCentrovacky.ResetStep:= TRUE;
				SC_OvlCentrovacky.Step:= 0;
			ELSIF SC_OvlCentrovacky.AlarmTime.Q THEN
				P34_Alarmy[304]:= TRUE;
				P3_Pracovisko.STAV.Porucha_ST6:= TRUE;
			END_IF

		20:
			SC_OvlCentrovacky.StepName:= '20 - Zasunutie centrovacky';
			SC_OvlCentrovacky.IdleTime.PT:= T#3s;
			SC_OvlCentrovacky.AlarmTime.PT:= T#10s;

			IF P3_LeakageTestB.Automat THEN
				SC_OvlCentrovacky.AlarmTime.IN:= TRUE;
			ELSE
				SC_OvlCentrovacky.IdleTime.IN:= TRUE;
			END_IF

			IF NOT SC_OvlCentrovacky.Switch1 THEN
				P3_LeakageTestB.OUT.Centrovanie_VYSUN:= FALSE;
                P3_LeakageTestB.OUT.PneuZamokCentrovania_ODOMKNI:= TRUE;
				SC_OvlCentrovacky.Switch1:= TRUE;
			END_IF

			IF P3_LeakageTestB.IN.Centrovanie_ZASUNUTE OR SC_OvlCentrovacky.IdleTime.Q THEN
				SC_OvlCentrovacky.ResetStep:= TRUE;
				SC_OvlCentrovacky.Step:= 0;
			ELSIF SC_OvlCentrovacky.AlarmTime.Q THEN
				P34_Alarmy[305]:= TRUE;
				P3_Pracovisko.STAV.Porucha_ST6:= TRUE;
			END_IF

	END_CASE

END_ACTION
```

#### OvlHornehoPritlaku.st
```iecst
ACTION OvlHornehoPritlaku:

	//Volanie funkcie SequenceControl//
	SequenceControl(SC:= SC_OvlHornehoPritlaku);

	CASE SC_OvlHornehoPritlaku.Step OF

		0:
			SC_OvlHornehoPritlaku.StepName:= '0 - Nulovanie';
			HornyPritlak_VYSUN:= FALSE;
			HornyPritlak_ZASUN:= FALSE;

			IF SC_P3_LeakageTestB.Step <> 0 THEN
				SC_OvlHornehoPritlaku.ResetStep:= TRUE;
				SC_OvlHornehoPritlaku.Step:= 1;
			END_IF

		1:
			SC_OvlHornehoPritlaku.StepName:= '1 - Rozhodnutie o cinnosti';
			IF HornyPritlak_VYSUN THEN
				SC_OvlHornehoPritlaku.Step:= 10;
			ELSIF HornyPritlak_ZASUN THEN
				SC_OvlHornehoPritlaku.Step:= 20;
			END_IF

		10:
			SC_OvlHornehoPritlaku.StepName:= '10 - Vysunutie horneho pritlaku';
			SC_OvlHornehoPritlaku.IdleTime.PT:= T#3s;
			SC_OvlHornehoPritlaku.AlarmTime.PT:= T#6s;

			IF P3_LeakageTestB.Automat THEN
				SC_OvlHornehoPritlaku.AlarmTime.IN:= TRUE;
			ELSE
				SC_OvlHornehoPritlaku.IdleTime.IN:= TRUE;
			END_IF

			IF NOT SC_OvlHornehoPritlaku.Switch1 THEN
				P3_LeakageTestB.OUT.PneuZamokZvonu_ODOMKNI:= TRUE;
				P3_LeakageTestB.OUT.HornyPritlak_ZASUN:= FALSE;
				P3_LeakageTestB.OUT.HornyPritlak_VYSUN:= TRUE;
				SC_OvlHornehoPritlaku.Switch1:= TRUE;
			END_IF

			IF P3_LeakageTestB.IN.HornyPritlak_VYSUNUTY OR SC_OvlHornehoPritlaku.IdleTime.Q THEN
				SC_OvlHornehoPritlaku.ResetStep:= TRUE;
				SC_OvlHornehoPritlaku.Step:= 0;
			ELSIF SC_OvlHornehoPritlaku.AlarmTime.Q THEN
				P34_Alarmy[308]:= TRUE;
				P3_Pracovisko.STAV.Porucha_ST6:= TRUE;
			END_IF

		20:
			SC_OvlHornehoPritlaku.StepName:= '20 - Zasunutie horneho pritlaku';
			SC_OvlHornehoPritlaku.IdleTime.PT:= T#3s;
			SC_OvlHornehoPritlaku.AlarmTime.PT:= T#6s;

			IF P3_LeakageTestB.Automat THEN
				SC_OvlHornehoPritlaku.AlarmTime.IN:= TRUE;
			ELSE
				SC_OvlHornehoPritlaku.IdleTime.IN:= TRUE;
			END_IF

			IF NOT SC_OvlHornehoPritlaku.Switch1 THEN
				P3_LeakageTestB.OUT.PneuZamokZvonu_ODOMKNI:= TRUE;
				P3_LeakageTestB.OUT.HornyPritlak_VYSUN:= FALSE;
				P3_LeakageTestB.OUT.HornyPritlak_ZASUN:= TRUE;
				SC_OvlHornehoPritlaku.Switch1:= TRUE;
			END_IF

			IF P3_LeakageTestB.IN.HornyPritlak_ZASUNUTY OR SC_OvlHornehoPritlaku.IdleTime.Q THEN
				SC_OvlHornehoPritlaku.ResetStep:= TRUE;
				SC_OvlHornehoPritlaku.Step:= 0;
			ELSIF SC_OvlHornehoPritlaku.AlarmTime.Q THEN
				P34_Alarmy[309]:= TRUE;
				P3_Pracovisko.STAV.Porucha_ST6:= TRUE;
			END_IF

	END_CASE

END_ACTION
```

#### COM_Tester.st
```iecst
ACTION COM_Tester:

	//Vstupy z Testera do PLC//
	AteqLeakageTester_B.Stav_RESET_DONE:= AteqLeakageTester_B.Profinet_PLC_INPUTS[1].0;
	AteqLeakageTester_B.Stav_START_DONE:= AteqLeakageTester_B.Profinet_PLC_INPUTS[1].1;
	AteqLeakageTester_B.Stav_ZmenaProgramu_DONE:= AteqLeakageTester_B.Profinet_PLC_INPUTS[1].3;
	AteqLeakageTester_B.Stav_CitanieParametrov_OK:= AteqLeakageTester_B.Profinet_PLC_INPUTS[1].5;

	AteqLeakageTester_B.Stav_CitanieParametrov_ERROR:= AteqLeakageTester_B.Profinet_PLC_INPUTS[3].5;

	AteqLeakageTester_B.CisloAktualnehoProgramu.0:= AteqLeakageTester_B.Profinet_PLC_INPUTS[7].0;
	AteqLeakageTester_B.CisloAktualnehoProgramu.1:= AteqLeakageTester_B.Profinet_PLC_INPUTS[7].1;
	AteqLeakageTester_B.CisloAktualnehoProgramu.2:= AteqLeakageTester_B.Profinet_PLC_INPUTS[7].2;
	AteqLeakageTester_B.CisloAktualnehoProgramu.3:= AteqLeakageTester_B.Profinet_PLC_INPUTS[7].3;
	AteqLeakageTester_B.CisloAktualnehoProgramu.4:= AteqLeakageTester_B.Profinet_PLC_INPUTS[7].4;
	AteqLeakageTester_B.CisloAktualnehoProgramu.5:= AteqLeakageTester_B.Profinet_PLC_INPUTS[7].5;
	AteqLeakageTester_B.CisloAktualnehoProgramu.6:= AteqLeakageTester_B.Profinet_PLC_INPUTS[7].6;
	AteqLeakageTester_B.CisloAktualnehoProgramu.7:= AteqLeakageTester_B.Profinet_PLC_INPUTS[7].7;

	AteqLeakageTester_B.CisloAktualnehoProgramu.8:= AteqLeakageTester_B.Profinet_PLC_INPUTS[8].0;
	AteqLeakageTester_B.CisloAktualnehoProgramu.9:= AteqLeakageTester_B.Profinet_PLC_INPUTS[8].1;
	AteqLeakageTester_B.CisloAktualnehoProgramu.10:= AteqLeakageTester_B.Profinet_PLC_INPUTS[8].2;
	AteqLeakageTester_B.CisloAktualnehoProgramu.11:= AteqLeakageTester_B.Profinet_PLC_INPUTS[8].3;
	AteqLeakageTester_B.CisloAktualnehoProgramu.12:= AteqLeakageTester_B.Profinet_PLC_INPUTS[8].4;
	AteqLeakageTester_B.CisloAktualnehoProgramu.13:= AteqLeakageTester_B.Profinet_PLC_INPUTS[8].5;
	AteqLeakageTester_B.CisloAktualnehoProgramu.14:= AteqLeakageTester_B.Profinet_PLC_INPUTS[8].6;
	AteqLeakageTester_B.CisloAktualnehoProgramu.15:= AteqLeakageTester_B.Profinet_PLC_INPUTS[8].7;

	AteqLeakageTester_B.VysledokTestovania_OK:= AteqLeakageTester_B.Profinet_PLC_INPUTS[13].0;
	AteqLeakageTester_B.VysledokTestovania_NG:= AteqLeakageTester_B.Profinet_PLC_INPUTS[13].1;
	AteqLeakageTester_B.Stav_ERROR:= AteqLeakageTester_B.Profinet_PLC_INPUTS[13].3;
	AteqLeakageTester_B.Stav_READY:= AteqLeakageTester_B.Profinet_PLC_INPUTS[13].5;

	AteqLeakageTester_B.ReadParameter_1.0:= AteqLeakageTester_B.Profinet_PLC_INPUTS[35].0;
	AteqLeakageTester_B.ReadParameter_1.1:= AteqLeakageTester_B.Profinet_PLC_INPUTS[35].1;
	AteqLeakageTester_B.ReadParameter_1.2:= AteqLeakageTester_B.Profinet_PLC_INPUTS[35].2;
	AteqLeakageTester_B.ReadParameter_1.3:= AteqLeakageTester_B.Profinet_PLC_INPUTS[35].3;
	AteqLeakageTester_B.ReadParameter_1.4:= AteqLeakageTester_B.Profinet_PLC_INPUTS[35].4;
	AteqLeakageTester_B.ReadParameter_1.5:= AteqLeakageTester_B.Profinet_PLC_INPUTS[35].5;
	AteqLeakageTester_B.ReadParameter_1.6:= AteqLeakageTester_B.Profinet_PLC_INPUTS[35].6;
	AteqLeakageTester_B.ReadParameter_1.7:= AteqLeakageTester_B.Profinet_PLC_INPUTS[35].7;
	AteqLeakageTester_B.ReadParameter_1.8:= AteqLeakageTester_B.Profinet_PLC_INPUTS[36].0;
	AteqLeakageTester_B.ReadParameter_1.9:= AteqLeakageTester_B.Profinet_PLC_INPUTS[36].1;
	AteqLeakageTester_B.ReadParameter_1.10:= AteqLeakageTester_B.Profinet_PLC_INPUTS[36].2;
	AteqLeakageTester_B.ReadParameter_1.11:= AteqLeakageTester_B.Profinet_PLC_INPUTS[36].3;
	AteqLeakageTester_B.ReadParameter_1.12:= AteqLeakageTester_B.Profinet_PLC_INPUTS[36].4;
	AteqLeakageTester_B.ReadParameter_1.13:= AteqLeakageTester_B.Profinet_PLC_INPUTS[36].5;
	AteqLeakageTester_B.ReadParameter_1.14:= AteqLeakageTester_B.Profinet_PLC_INPUTS[36].6;
	AteqLeakageTester_B.ReadParameter_1.15:= AteqLeakageTester_B.Profinet_PLC_INPUTS[36].7;

	AteqLeakageTester_B.ReadParameter_2.0:= AteqLeakageTester_B.Profinet_PLC_INPUTS[41].0;
	AteqLeakageTester_B.ReadParameter_2.1:= AteqLeakageTester_B.Profinet_PLC_INPUTS[41].1;
	AteqLeakageTester_B.ReadParameter_2.2:= AteqLeakageTester_B.Profinet_PLC_INPUTS[41].2;
	AteqLeakageTester_B.ReadParameter_2.3:= AteqLeakageTester_B.Profinet_PLC_INPUTS[41].3;
	AteqLeakageTester_B.ReadParameter_2.4:= AteqLeakageTester_B.Profinet_PLC_INPUTS[41].4;
	AteqLeakageTester_B.ReadParameter_2.5:= AteqLeakageTester_B.Profinet_PLC_INPUTS[41].5;
	AteqLeakageTester_B.ReadParameter_2.6:= AteqLeakageTester_B.Profinet_PLC_INPUTS[41].6;
	AteqLeakageTester_B.ReadParameter_2.7:= AteqLeakageTester_B.Profinet_PLC_INPUTS[41].7;
	AteqLeakageTester_B.ReadParameter_2.8:= AteqLeakageTester_B.Profinet_PLC_INPUTS[42].0;
	AteqLeakageTester_B.ReadParameter_2.9:= AteqLeakageTester_B.Profinet_PLC_INPUTS[42].1;
	AteqLeakageTester_B.ReadParameter_2.10:= AteqLeakageTester_B.Profinet_PLC_INPUTS[42].2;
	AteqLeakageTester_B.ReadParameter_2.11:= AteqLeakageTester_B.Profinet_PLC_INPUTS[42].3;
	AteqLeakageTester_B.ReadParameter_2.12:= AteqLeakageTester_B.Profinet_PLC_INPUTS[42].4;
	AteqLeakageTester_B.ReadParameter_2.13:= AteqLeakageTester_B.Profinet_PLC_INPUTS[42].5;
	AteqLeakageTester_B.ReadParameter_2.14:= AteqLeakageTester_B.Profinet_PLC_INPUTS[42].6;
	AteqLeakageTester_B.ReadParameter_2.15:= AteqLeakageTester_B.Profinet_PLC_INPUTS[42].7;

	AteqLeakageTester_B.ReadParameter_3.0:= AteqLeakageTester_B.Profinet_PLC_INPUTS[47].0;
	AteqLeakageTester_B.ReadParameter_3.1:= AteqLeakageTester_B.Profinet_PLC_INPUTS[47].1;
	AteqLeakageTester_B.ReadParameter_3.2:= AteqLeakageTester_B.Profinet_PLC_INPUTS[47].2;
	AteqLeakageTester_B.ReadParameter_3.3:= AteqLeakageTester_B.Profinet_PLC_INPUTS[47].3;
	AteqLeakageTester_B.ReadParameter_3.4:= AteqLeakageTester_B.Profinet_PLC_INPUTS[47].4;
	AteqLeakageTester_B.ReadParameter_3.5:= AteqLeakageTester_B.Profinet_PLC_INPUTS[47].5;
	AteqLeakageTester_B.ReadParameter_3.6:= AteqLeakageTester_B.Profinet_PLC_INPUTS[47].6;
	AteqLeakageTester_B.ReadParameter_3.7:= AteqLeakageTester_B.Profinet_PLC_INPUTS[47].7;
	AteqLeakageTester_B.ReadParameter_3.8:= AteqLeakageTester_B.Profinet_PLC_INPUTS[48].0;
	AteqLeakageTester_B.ReadParameter_3.9:= AteqLeakageTester_B.Profinet_PLC_INPUTS[48].1;
	AteqLeakageTester_B.ReadParameter_3.10:= AteqLeakageTester_B.Profinet_PLC_INPUTS[48].2;
	AteqLeakageTester_B.ReadParameter_3.11:= AteqLeakageTester_B.Profinet_PLC_INPUTS[48].3;
	AteqLeakageTester_B.ReadParameter_3.12:= AteqLeakageTester_B.Profinet_PLC_INPUTS[48].4;
	AteqLeakageTester_B.ReadParameter_3.13:= AteqLeakageTester_B.Profinet_PLC_INPUTS[48].5;
	AteqLeakageTester_B.ReadParameter_3.14:= AteqLeakageTester_B.Profinet_PLC_INPUTS[48].6;
	AteqLeakageTester_B.ReadParameter_3.15:= AteqLeakageTester_B.Profinet_PLC_INPUTS[48].7;

	AteqLeakageTester_B.ReadParameter_4.0:= AteqLeakageTester_B.Profinet_PLC_INPUTS[53].0;
	AteqLeakageTester_B.ReadParameter_4.1:= AteqLeakageTester_B.Profinet_PLC_INPUTS[53].1;
	AteqLeakageTester_B.ReadParameter_4.2:= AteqLeakageTester_B.Profinet_PLC_INPUTS[53].2;
	AteqLeakageTester_B.ReadParameter_4.3:= AteqLeakageTester_B.Profinet_PLC_INPUTS[53].3;
	AteqLeakageTester_B.ReadParameter_4.4:= AteqLeakageTester_B.Profinet_PLC_INPUTS[53].4;
	AteqLeakageTester_B.ReadParameter_4.5:= AteqLeakageTester_B.Profinet_PLC_INPUTS[53].5;
	AteqLeakageTester_B.ReadParameter_4.6:= AteqLeakageTester_B.Profinet_PLC_INPUTS[53].6;
	AteqLeakageTester_B.ReadParameter_4.7:= AteqLeakageTester_B.Profinet_PLC_INPUTS[53].7;
	AteqLeakageTester_B.ReadParameter_4.8:= AteqLeakageTester_B.Profinet_PLC_INPUTS[54].0;
	AteqLeakageTester_B.ReadParameter_4.9:= AteqLeakageTester_B.Profinet_PLC_INPUTS[54].1;
	AteqLeakageTester_B.ReadParameter_4.10:= AteqLeakageTester_B.Profinet_PLC_INPUTS[54].2;
	AteqLeakageTester_B.ReadParameter_4.11:= AteqLeakageTester_B.Profinet_PLC_INPUTS[54].3;
	AteqLeakageTester_B.ReadParameter_4.12:= AteqLeakageTester_B.Profinet_PLC_INPUTS[54].4;
	AteqLeakageTester_B.ReadParameter_4.13:= AteqLeakageTester_B.Profinet_PLC_INPUTS[54].5;
	AteqLeakageTester_B.ReadParameter_4.14:= AteqLeakageTester_B.Profinet_PLC_INPUTS[54].6;
	AteqLeakageTester_B.ReadParameter_4.15:= AteqLeakageTester_B.Profinet_PLC_INPUTS[54].7;

	AteqLeakageTester_B.ReadParameter_5.0:= AteqLeakageTester_B.Profinet_PLC_INPUTS[24].0;
	AteqLeakageTester_B.ReadParameter_5.1:= AteqLeakageTester_B.Profinet_PLC_INPUTS[24].1;
	AteqLeakageTester_B.ReadParameter_5.2:= AteqLeakageTester_B.Profinet_PLC_INPUTS[24].2;
	AteqLeakageTester_B.ReadParameter_5.3:= AteqLeakageTester_B.Profinet_PLC_INPUTS[24].3;
	AteqLeakageTester_B.ReadParameter_5.4:= AteqLeakageTester_B.Profinet_PLC_INPUTS[24].4;
	AteqLeakageTester_B.ReadParameter_5.5:= AteqLeakageTester_B.Profinet_PLC_INPUTS[24].5;
	AteqLeakageTester_B.ReadParameter_5.6:= AteqLeakageTester_B.Profinet_PLC_INPUTS[24].6;
	AteqLeakageTester_B.ReadParameter_5.7:= AteqLeakageTester_B.Profinet_PLC_INPUTS[24].7;
	AteqLeakageTester_B.ReadParameter_5.8:= AteqLeakageTester_B.Profinet_PLC_INPUTS[25].0;
	AteqLeakageTester_B.ReadParameter_5.9:= AteqLeakageTester_B.Profinet_PLC_INPUTS[25].1;
	AteqLeakageTester_B.ReadParameter_5.10:= AteqLeakageTester_B.Profinet_PLC_INPUTS[25].2;
	AteqLeakageTester_B.ReadParameter_5.11:= AteqLeakageTester_B.Profinet_PLC_INPUTS[25].3;
	AteqLeakageTester_B.ReadParameter_5.12:= AteqLeakageTester_B.Profinet_PLC_INPUTS[25].4;
	AteqLeakageTester_B.ReadParameter_5.13:= AteqLeakageTester_B.Profinet_PLC_INPUTS[25].5;
	AteqLeakageTester_B.ReadParameter_5.14:= AteqLeakageTester_B.Profinet_PLC_INPUTS[25].6;
	AteqLeakageTester_B.ReadParameter_5.15:= AteqLeakageTester_B.Profinet_PLC_INPUTS[25].7;
	AteqLeakageTester_B.ReadParameter_5.16:= AteqLeakageTester_B.Profinet_PLC_INPUTS[26].0;
	AteqLeakageTester_B.ReadParameter_5.17:= AteqLeakageTester_B.Profinet_PLC_INPUTS[26].1;
	AteqLeakageTester_B.ReadParameter_5.18:= AteqLeakageTester_B.Profinet_PLC_INPUTS[26].2;
	AteqLeakageTester_B.ReadParameter_5.19:= AteqLeakageTester_B.Profinet_PLC_INPUTS[26].3;
	AteqLeakageTester_B.ReadParameter_5.20:= AteqLeakageTester_B.Profinet_PLC_INPUTS[26].4;
	AteqLeakageTester_B.ReadParameter_5.21:= AteqLeakageTester_B.Profinet_PLC_INPUTS[26].5;
	AteqLeakageTester_B.ReadParameter_5.22:= AteqLeakageTester_B.Profinet_PLC_INPUTS[26].6;
	AteqLeakageTester_B.ReadParameter_5.23:= AteqLeakageTester_B.Profinet_PLC_INPUTS[26].7;
	AteqLeakageTester_B.ReadParameter_5.24:= AteqLeakageTester_B.Profinet_PLC_INPUTS[27].0;
	AteqLeakageTester_B.ReadParameter_5.25:= AteqLeakageTester_B.Profinet_PLC_INPUTS[27].1;
	AteqLeakageTester_B.ReadParameter_5.26:= AteqLeakageTester_B.Profinet_PLC_INPUTS[27].2;
	AteqLeakageTester_B.ReadParameter_5.27:= AteqLeakageTester_B.Profinet_PLC_INPUTS[27].3;
	AteqLeakageTester_B.ReadParameter_5.28:= AteqLeakageTester_B.Profinet_PLC_INPUTS[27].4;
	AteqLeakageTester_B.ReadParameter_5.29:= AteqLeakageTester_B.Profinet_PLC_INPUTS[27].5;
	AteqLeakageTester_B.ReadParameter_5.30:= AteqLeakageTester_B.Profinet_PLC_INPUTS[27].6;
	AteqLeakageTester_B.ReadParameter_5.31:= AteqLeakageTester_B.Profinet_PLC_INPUTS[27].7;

	//Vystupy z PLC do Testera//
	AteqLeakageTester_B.Profinet_PLC_OUTPUTS[1].0:= AteqLeakageTester_B.RESET_Vysledkov;
	AteqLeakageTester_B.Profinet_PLC_OUTPUTS[1].1:= AteqLeakageTester_B.START_Testovania;
	AteqLeakageTester_B.Profinet_PLC_OUTPUTS[1].3:= AteqLeakageTester_B.ZMEN_Program;
	AteqLeakageTester_B.Profinet_PLC_OUTPUTS[1].5:= AteqLeakageTester_B.CitajParametreTestera;

	AteqLeakageTester_B.Profinet_PLC_OUTPUTS[7].0:= AteqLeakageTester_B.CisloZadanehoProgramu.0;
	AteqLeakageTester_B.Profinet_PLC_OUTPUTS[7].1:= AteqLeakageTester_B.CisloZadanehoProgramu.1;
	AteqLeakageTester_B.Profinet_PLC_OUTPUTS[7].2:= AteqLeakageTester_B.CisloZadanehoProgramu.2;
	AteqLeakageTester_B.Profinet_PLC_OUTPUTS[7].3:= AteqLeakageTester_B.CisloZadanehoProgramu.3;
	AteqLeakageTester_B.Profinet_PLC_OUTPUTS[7].4:= AteqLeakageTester_B.CisloZadanehoProgramu.4;
	AteqLeakageTester_B.Profinet_PLC_OUTPUTS[7].5:= AteqLeakageTester_B.CisloZadanehoProgramu.5;
	AteqLeakageTester_B.Profinet_PLC_OUTPUTS[7].6:= AteqLeakageTester_B.CisloZadanehoProgramu.6;
	AteqLeakageTester_B.Profinet_PLC_OUTPUTS[7].7:= AteqLeakageTester_B.CisloZadanehoProgramu.7;

	AteqLeakageTester_B.Profinet_PLC_OUTPUTS[8].0:= AteqLeakageTester_B.CisloZadanehoProgramu.8;
	AteqLeakageTester_B.Profinet_PLC_OUTPUTS[8].1:= AteqLeakageTester_B.CisloZadanehoProgramu.9;
	AteqLeakageTester_B.Profinet_PLC_OUTPUTS[8].2:= AteqLeakageTester_B.CisloZadanehoProgramu.10;
	AteqLeakageTester_B.Profinet_PLC_OUTPUTS[8].3:= AteqLeakageTester_B.CisloZadanehoProgramu.11;
	AteqLeakageTester_B.Profinet_PLC_OUTPUTS[8].4:= AteqLeakageTester_B.CisloZadanehoProgramu.12;
	AteqLeakageTester_B.Profinet_PLC_OUTPUTS[8].5:= AteqLeakageTester_B.CisloZadanehoProgramu.13;
	AteqLeakageTester_B.Profinet_PLC_OUTPUTS[8].6:= AteqLeakageTester_B.CisloZadanehoProgramu.14;
	AteqLeakageTester_B.Profinet_PLC_OUTPUTS[8].7:= AteqLeakageTester_B.CisloZadanehoProgramu.15;

	AteqLeakageTester_B.PocetCitanychParametrov:= 4;
	AteqLeakageTester_B.IdentifikaciaParametra_1:= 1;
	AteqLeakageTester_B.IdentifikaciaParametra_2:= 2;
	AteqLeakageTester_B.IdentifikaciaParametra_3:= 66;
	AteqLeakageTester_B.IdentifikaciaParametra_4:= 60;

	//Vyčítané parametre//
	CasPneniaREAL:= UINT_TO_REAL(AteqLeakageTester_B.ReadParameter_1);
	AteqLeakageTester_B.CasPnenia:= CasPneniaREAL/1000;
	CasStabilizacieREAL:= UINT_TO_REAL(AteqLeakageTester_B.ReadParameter_2);
	AteqLeakageTester_B.CasStabilizacie:= CasStabilizacieREAL/1000;
	TlakPlneniaREAL:= UINT_TO_REAL(AteqLeakageTester_B.ReadParameter_3);
	AteqLeakageTester_B.TlakPlnenia:= TlakPlneniaREAL/1000;
	ToleranciaREAL:= UINT_TO_REAL(AteqLeakageTester_B.ReadParameter_4);
	AteqLeakageTester_B.Tolerancia:= ToleranciaREAL/1000;
	TlakUnikuREAL:= DINT_TO_REAL(AteqLeakageTester_B.ReadParameter_5);
	AteqLeakageTester_B.TlakUniku:= ((TlakUnikuREAL/1000)*6)/1536;

END_ACTION
```

### Program Logical/Program/Pracovisko_3/P3_ZdvizkaZaLeakTestA (IEC)

#### Main.st - Init, cyclic, exit code
```iecst
PROGRAM _INIT
	(* Insert code here *)

END_PROGRAM

PROGRAM _CYCLIC

	//Volanie funkcie SequenceControl//
	SequenceControl(SC:= SC_P3_ZdvizkaZaLeakTestA);

	//Volanie podprogramov//
	OvlZdvizky;

	//Reset sekcie //
	IF P3_ZdvizkaZaLeakTestA.Reset THEN
		SC_P3_ZdvizkaZaLeakTestA.Step:= 0;
		P3_ZdvizkaZaLeakTestA.Reset:= FALSE;
	ELSIF NOT Safety.STAV.Linka_ZonaCS_AKTIVNA THEN
		SC_P3_ZdvizkaZaLeakTestA.Step:= 0;
	END_IF

	CASE SC_P3_ZdvizkaZaLeakTestA.Step OF

		0:
			SC_P3_ZdvizkaZaLeakTestA.StepName:='0 - Nulovanie';
			SC_OvlZdvizky.Step:= 0;
			P3_ZdvizkaZaLeakTestA.Automat:= FALSE;
			P3_ZdvizkaZaLeakTestA.KoniecCyklu:= FALSE;
			P3_ZdvizkaZaLeakTestA.Manual:= FALSE;
			P3_ZdvizkaZaLeakTestA.STAV.PoINIT:= FALSE;
			P3_ZdvizkaZaLeakTestA.OUT.TlmicPaletky_VYSUN:= FALSE;
			P3_ZdvizkaZaLeakTestA.OUT.TlmicPaletky_ZASUN:= FALSE;
			P3_Dopravniky.OUT.PriecnyDopravnik2_VPRED:= FALSE;
			P3_Dopravniky.OUT.PriecnyDopravnik2_VZAD:= FALSE;
			P3_ZdvizkaZaLeakTestA.STAV.PrebiehaVyvezeniePaletkyNaTratA:= FALSE;
			P3_ZdvizkaZaLeakTestA.STAV.PrebiehaVyvezeniePaletkyNaTratB:= FALSE;
			P3_LeakageTestA.STAV.PrebiehaVyvezeniePaletky:= FALSE;

			IF Safety.STAV.Linka_ZonaCS_AKTIVNA AND
				Safety.STAV.P3_ZonaBunky_AKTIVNA AND
				P3_Pracovisko.STAV.HardwareBunky_OK AND
				NOT P3_Pracovisko.STAV.Porucha_ST1 AND
				NOT P3_Pracovisko.STAV.Porucha_ST2 AND
				NOT P3_Pracovisko.STAV.Porucha_ST3 AND
				NOT P3_Pracovisko.STAV.Porucha_ST4 AND
				NOT P3_Pracovisko.STAV.Porucha_ST5 AND
				NOT P3_Pracovisko.STAV.Porucha_ST6 AND
				NOT P3_Pracovisko.STAV.Porucha_ST7 AND
				NOT P3_Pracovisko.STAV.Porucha_ST8 THEN
				SC_P3_ZdvizkaZaLeakTestA.ResetStep:= TRUE;
				SC_P3_ZdvizkaZaLeakTestA.Step:= 1;
			END_IF

		1:
			SC_P3_ZdvizkaZaLeakTestA.StepName:='1 - Cakam na spustenie vyroby';
			P3_ZdvizkaZaLeakTestA.KoniecCyklu:= FALSE;
			IF P3_ZdvizkaZaLeakTestA.Automat THEN
				SC_P3_ZdvizkaZaLeakTestA.Step:= 2;
			ELSIF P3_ZdvizkaZaLeakTestA.Manual THEN
				SC_P3_ZdvizkaZaLeakTestA.Step:= 700;
			END_IF

			//********************************************************Inicializácia****************************************************************************//

		2:
			SC_P3_ZdvizkaZaLeakTestA.StepName:='2 - Inicializacia - cakam na spustenie inicializacie';
			SC_P3_ZdvizkaZaLeakTestA.IdleTime.PT:= T#500ms;
			SC_P3_ZdvizkaZaLeakTestA.AlarmTime.PT:= T#5s;

			IF P3_Dopravniky.STAV.PoINIT AND P3_ZdvizkaZaLeakTestB.STAV.PoINIT THEN
				SC_P3_ZdvizkaZaLeakTestA.ResetStep:= TRUE;
				SC_P3_ZdvizkaZaLeakTestA.Step:= 5;
			END_IF

		5:
			SC_P3_ZdvizkaZaLeakTestA.StepName:='5 - Inicializacia - kontrola pozicie zdvizky';
			SC_P3_ZdvizkaZaLeakTestA.IdleTime.PT:= T#500ms;
			SC_P3_ZdvizkaZaLeakTestA.AlarmTime.PT:= T#5s;

			IF P3_ZdvizkaZaLeakTestA.IN.Zdvizka_StrednaPoloha AND P3_ZdvizkaZaLeakTestA.IN.PritomnostPaletky THEN
				P3_ZdvizkaZaLeakTestA.STAV.PoINIT:= TRUE;
				SC_P3_ZdvizkaZaLeakTestA.ResetStep:= TRUE;
				SC_P3_ZdvizkaZaLeakTestA.Step:= 100;
			ELSE
				SC_P3_ZdvizkaZaLeakTestA.ResetStep:= TRUE;
				SC_P3_ZdvizkaZaLeakTestA.Step:= 8;
			END_IF

		8:
			SC_P3_ZdvizkaZaLeakTestA.StepName:='8 - Inicializacia - presun zdvizky do hornej polohy';
			SC_P3_ZdvizkaZaLeakTestA.IdleTime.PT:= T#5s;
			SC_P3_ZdvizkaZaLeakTestA.AlarmTime.PT:= T#5s;

			IF NOT SC_P3_ZdvizkaZaLeakTestA.Switch1 AND SC_OvlZdvizky.Step = 1 THEN
				Zdvizku_VYSUN:= TRUE;
				P3_ZdvizkaZaLeakTestA.OUT.TlmicPaletky_VYSUN:= FALSE;
				P3_ZdvizkaZaLeakTestA.OUT.TlmicPaletky_ZASUN:= TRUE;
				SC_P3_ZdvizkaZaLeakTestA.Switch1:= TRUE;
			END_IF

			IF P3_ZdvizkaZaLeakTestA.IN.Zdvizka_HornaPoloha AND P3_ZdvizkaZaLeakTestA.IN.TlmicPaletky_ZASUNUTY THEN
				SC_P3_ZdvizkaZaLeakTestA.ResetStep:= TRUE;
				SC_P3_ZdvizkaZaLeakTestA.Step:= 10;
			END_IF

		10:
			SC_P3_ZdvizkaZaLeakTestA.StepName:='10 - Inicializacia - kontrola pritomnosti paletky na zdvizke za Leakage Testom B';
			SC_P3_ZdvizkaZaLeakTestA.IdleTime.PT:= T#500ms;
			SC_P3_ZdvizkaZaLeakTestA.AlarmTime.PT:= T#5s;

			IF NOT P3_ZdvizkaZaLeakTestB.IN.PritomnostPaletky THEN
				P3_ZdvizkaZaLeakTestB.OUT.Zdvizku_ZASUN:= FALSE;
				P3_ZdvizkaZaLeakTestB.OUT.Zdvizku_VYSUN:= TRUE;
				SC_P3_ZdvizkaZaLeakTestA.ResetStep:= TRUE;
				SC_P3_ZdvizkaZaLeakTestA.Step:= 11;
			ELSE
				SC_P3_ZdvizkaZaLeakTestA.ResetStep:= TRUE;
				SC_P3_ZdvizkaZaLeakTestA.Step:= 13;
			END_IF

		11:
			SC_P3_ZdvizkaZaLeakTestA.StepName:='11 - Inicializacia - cakam na zodvihnutie zdvizky za Leakage Testom B';
			SC_P3_ZdvizkaZaLeakTestA.IdleTime.PT:= T#500ms;
			SC_P3_ZdvizkaZaLeakTestA.AlarmTime.PT:= T#5s;

			IF P3_ZdvizkaZaLeakTestB.IN.Zdvizka_HornaPoloha THEN
				SC_P3_ZdvizkaZaLeakTestA.ResetStep:= TRUE;
				SC_P3_ZdvizkaZaLeakTestA.Step:= 13;
			END_IF

		13:
			SC_P3_ZdvizkaZaLeakTestA.StepName:='13 - Inicializacia - spustenie priecneho dopravnika';
			SC_P3_ZdvizkaZaLeakTestA.IdleTime.PT:= T#500ms;
			SC_P3_ZdvizkaZaLeakTestA.AlarmTime.PT:= T#7s;

			SC_P3_ZdvizkaZaLeakTestA.IdleTime.IN:= P3_ZdvizkaZaLeakTestA.IN.PritomnostPaletky AND P3_ZdvizkaZaLeakTestA.IN.PoziciaPaletky_OK;

			IF NOT SC_P3_ZdvizkaZaLeakTestA.Switch1 THEN
				P3_Dopravniky.OUT.PriecnyDopravnik2_VPRED:= FALSE;
				P3_Dopravniky.OUT.PriecnyDopravnik2_VZAD:= TRUE;
				SC_P3_ZdvizkaZaLeakTestA.AlarmTime.IN:= TRUE;
				SC_P3_ZdvizkaZaLeakTestA.Switch1:= TRUE;
			END_IF

			IF SC_P3_ZdvizkaZaLeakTestA.IdleTime.Q THEN
				P3_Dopravniky.OUT.PriecnyDopravnik2_VZAD:= FALSE;
				P3_Dopravniky.OUT.PriecnyDopravnik2_VPRED:= FALSE;
				SC_P3_ZdvizkaZaLeakTestA.ResetStep:= TRUE;
				SC_P3_ZdvizkaZaLeakTestA.Step:= 15;
			ELSIF SC_P3_ZdvizkaZaLeakTestA.AlarmTime.Q THEN
				P3_Dopravniky.OUT.PriecnyDopravnik2_VZAD:= FALSE;
				P3_Dopravniky.OUT.PriecnyDopravnik2_VPRED:= FALSE;
				SC_P3_ZdvizkaZaLeakTestA.ResetStep:= TRUE;
				SC_P3_ZdvizkaZaLeakTestA.Step:= 15;
			END_IF

		15:
			SC_P3_ZdvizkaZaLeakTestA.StepName:='15 - Inicializacia - presun zdvizky do strednej polohy';
			SC_P3_ZdvizkaZaLeakTestA.IdleTime.PT:= T#500ms;
			SC_P3_ZdvizkaZaLeakTestA.AlarmTime.PT:= T#5s;

			IF NOT SC_P3_ZdvizkaZaLeakTestA.Switch1 AND SC_OvlZdvizky.Step = 1 THEN
				Zdvizku_VYSTRED:= TRUE;
				P3_ZdvizkaZaLeakTestB.OUT.Zdvizku_ZASUN:= FALSE;
				P3_ZdvizkaZaLeakTestB.OUT.Zdvizku_VYSUN:= FALSE;
				SC_P3_ZdvizkaZaLeakTestA.Switch1:= TRUE;
			END_IF

			IF P3_ZdvizkaZaLeakTestA.IN.Zdvizka_StrednaPoloha AND P3_ZdvizkaZaLeakTestB.IN.Zdvizka_StrednaPoloha THEN
				IF P3_ZdvizkaZaLeakTestA.IN.PritomnostPaletky THEN
					P3_ZdvizkaZaLeakTestA.STAV.PoINIT:= TRUE;
					SC_P3_ZdvizkaZaLeakTestA.ResetStep:= TRUE;
					SC_P3_ZdvizkaZaLeakTestA.Step:= 100;
				ELSE
					SC_P3_ZdvizkaZaLeakTestA.ResetStep:= TRUE;
					SC_P3_ZdvizkaZaLeakTestA.Step:= 18;
				END_IF
			END_IF

		18:
			SC_P3_ZdvizkaZaLeakTestA.StepName:='18 - Inicializacia - vysunutie tlmica paletky';
			SC_P3_ZdvizkaZaLeakTestA.IdleTime.PT:= T#500ms;
			SC_P3_ZdvizkaZaLeakTestA.AlarmTime.PT:= T#5s;

			IF NOT SC_P3_ZdvizkaZaLeakTestA.Switch1 THEN
				P3_ZdvizkaZaLeakTestA.OUT.TlmicPaletky_ZASUN:= FALSE;
				P3_ZdvizkaZaLeakTestA.OUT.TlmicPaletky_VYSUN:= TRUE;
				SC_P3_ZdvizkaZaLeakTestA.IdleTime.IN:= TRUE;
				SC_P3_ZdvizkaZaLeakTestA.Switch1:= TRUE;
			END_IF

			IF SC_P3_ZdvizkaZaLeakTestA.IdleTime.Q THEN
				P3_ZdvizkaZaLeakTestA.OUT.TlmicPaletky_ZASUN:= FALSE;
				P3_ZdvizkaZaLeakTestA.OUT.TlmicPaletky_VYSUN:= FALSE;
				P3_ZdvizkaZaLeakTestA.STAV.PoINIT:= TRUE;
				SC_P3_ZdvizkaZaLeakTestA.ResetStep:= TRUE;
				SC_P3_ZdvizkaZaLeakTestA.Step:= 100;
			END_IF

			//********************************************************Automatický režim****************************************************************************//

		100:
			SC_P3_ZdvizkaZaLeakTestA.StepName:='100 - Automaticky Rezim - cakam na príchod paletky na zdvizku';
			SC_P3_ZdvizkaZaLeakTestA.IdleTime.PT:= T#200ms;
			SC_P3_ZdvizkaZaLeakTestA.AlarmTime.PT:= T#5s;

			SC_P3_ZdvizkaZaLeakTestA.IdleTime.IN:= P3_ZdvizkaZaLeakTestA.IN.PritomnostPaletky AND P3_ZdvizkaZaLeakTestA.IN.PoziciaPaletky_OK AND P3_ZdvizkaZaLeakTestA.IN.TlmicPaletky_ZASUNUTY AND P3_ZdvizkaZaLeakTestA.IN.Zdvizka_StrednaPoloha;

			IF P3_ZdvizkaZaLeakTestA.IN.PritomnostPaletky AND P3_ZdvizkaZaLeakTestA.IN.Zdvizka_StrednaPoloha THEN
				P3_LeakageTestA.STAV.PrebiehaVyvezeniePaletky:= FALSE;
				P3_ZdvizkaZaLeakTestB.STAV.PrebiehaVyvezeniePaletkyNaTratA:= FALSE;
			END_IF

			IF P3_ZdvizkaZaLeakTestA.KoniecCyklu AND NOT P3_LeakageTestA.Automat THEN
				SC_P3_ZdvizkaZaLeakTestA.ResetStep:= TRUE;
				SC_P3_ZdvizkaZaLeakTestA.Step:= 0;
			ELSIF SC_P3_ZdvizkaZaLeakTestA.IdleTime.Q THEN
				SC_P3_ZdvizkaZaLeakTestA.ResetStep:= TRUE;
				SC_P3_ZdvizkaZaLeakTestA.Step:= 101;
			END_IF

		101:
			SC_P3_ZdvizkaZaLeakTestA.StepName:='101 - Automaticky Rezim - rozhodnutie o smere vyvazania';
			SC_P3_ZdvizkaZaLeakTestA.IdleTime.PT:= T#200ms;
			SC_P3_ZdvizkaZaLeakTestA.AlarmTime.PT:= T#5s;

			IF P3_ZdvizkaZaLeakTestA.KoniecCyklu AND NOT P3_LeakageTestA.Automat THEN
				SC_P3_ZdvizkaZaLeakTestA.ResetStep:= TRUE;
				SC_P3_ZdvizkaZaLeakTestA.Step:= 0;
			ELSIF P4_FunkcnyTestA.STAV.Tester_ON AND   //Vyvezenie na trať A//
				NOT P4_FunkcnyTestA.RFID_hlava.PritomnostPaletky AND
				SC_P4_FunkcnyTestA.Step = 100 AND
				NOT P3_ZdvizkaZaLeakTestA.STAV.PrebiehaVyvezeniePaletkyNaTratA AND
				NOT P3_ZdvizkaZaLeakTestB.STAV.PrebiehaVyvezeniePaletkyNaTratA THEN
				SC_P3_ZdvizkaZaLeakTestA.ResetStep:= TRUE;
				SC_P3_ZdvizkaZaLeakTestA.Step:= 110;
			ELSIF NOT P4_FunkcnyTestA.STAV.Tester_ON AND       //Vyvezenie na trať B//
				P4_FunkcnyTestB.STAV.Tester_ON AND
				NOT P3_ZdvizkaZaLeakTestB.IN.PritomnostPaletky AND
				SC_P3_ZdvizkaZaLeakTestB.Step = 100 AND
				NOT P3_ZdvizkaZaLeakTestB.STAV.PrebiehaVyvezeniePaletkyNaTratA AND
				NOT P3_LeakageTestB.STAV.PrebiehaVyvezeniePaletky AND
				SC_P3_LeakageTestB.Step < 560 THEN
				SC_P3_ZdvizkaZaLeakTestA.ResetStep:= TRUE;
				SC_P3_ZdvizkaZaLeakTestA.Step:= 120;
			ELSIF NOT P3_ZdvizkaZaLeakTestA.IN.PritomnostPaletky THEN
				SC_P3_ZdvizkaZaLeakTestA.ResetStep:= TRUE;
				SC_P3_ZdvizkaZaLeakTestA.Step:= 100;
			END_IF

			//Vyvážanie na trať A//
		110:
			SC_P3_ZdvizkaZaLeakTestA.StepName:='110 - Automaticky Rezim - presun zdvizky do spodnej polohy';
			SC_P3_ZdvizkaZaLeakTestA.IdleTime.PT:= T#200ms;
			SC_P3_ZdvizkaZaLeakTestA.AlarmTime.PT:= T#5s;

			IF NOT SC_P3_ZdvizkaZaLeakTestA.Switch1 AND SC_OvlZdvizky.Step = 1 THEN
				Zdvizku_ZASUN:= TRUE;
				P3_ZdvizkaZaLeakTestA.STAV.PrebiehaVyvezeniePaletkyNaTratA:= TRUE;
				SC_P3_ZdvizkaZaLeakTestA.Switch1:= TRUE;
			END_IF

			IF P3_ZdvizkaZaLeakTestA.IN.Zdvizka_SpodnaPoloha THEN
				SC_P3_ZdvizkaZaLeakTestA.ResetStep:= TRUE;
				SC_P3_ZdvizkaZaLeakTestA.Step:= 113;
			END_IF

		113:
			SC_P3_ZdvizkaZaLeakTestA.StepName:='113 - Automaticky Rezim - cakam na ukoncenie vyvazania na Trat A';
			SC_P3_ZdvizkaZaLeakTestA.IdleTime.PT:= T#500ms;
			SC_P3_ZdvizkaZaLeakTestA.AlarmTime.PT:= T#5s;

			SC_P3_ZdvizkaZaLeakTestA.IdleTime.IN:= NOT P3_ZdvizkaZaLeakTestA.IN.PritomnostPaletky;

			IF SC_P3_ZdvizkaZaLeakTestA.IdleTime.Q AND NOT SC_P3_ZdvizkaZaLeakTestA.Switch1 AND SC_OvlZdvizky.Step = 1 THEN
				Zdvizku_VYSTRED:= TRUE;
				SC_P3_ZdvizkaZaLeakTestA.Switch1:= TRUE;
			END_IF

			IF P3_ZdvizkaZaLeakTestA.IN.Zdvizka_StrednaPoloha THEN
				SC_P3_ZdvizkaZaLeakTestA.ResetStep:= TRUE;
				SC_P3_ZdvizkaZaLeakTestA.Step:= 130;
			END_IF

			//Vyvážanie na trať B//
		120:
			SC_P3_ZdvizkaZaLeakTestA.StepName:='120 - Automaticky Rezim - presun zdviziek do hornej polohy';
			SC_P3_ZdvizkaZaLeakTestA.IdleTime.PT:= T#200ms;
			SC_P3_ZdvizkaZaLeakTestA.AlarmTime.PT:= T#5s;

			IF NOT SC_P3_ZdvizkaZaLeakTestA.Switch1 AND SC_OvlZdvizky.Step = 1 THEN
				Zdvizku_VYSUN:= TRUE;
				P3_ZdvizkaZaLeakTestB.OUT.Zdvizku_ZASUN:= FALSE;
				P3_ZdvizkaZaLeakTestB.OUT.Zdvizku_VYSUN:= TRUE;
				P3_ZdvizkaZaLeakTestB.OUT.TlmicPaletky_VYSUN:= FALSE;
				P3_ZdvizkaZaLeakTestB.OUT.TlmicPaletky_ZASUN:= TRUE;
				P3_ZdvizkaZaLeakTestA.STAV.PrebiehaVyvezeniePaletkyNaTratB:= TRUE;
				SC_P3_ZdvizkaZaLeakTestA.Switch1:= TRUE;
			END_IF

			IF P3_ZdvizkaZaLeakTestA.IN.Zdvizka_HornaPoloha AND P3_ZdvizkaZaLeakTestB.IN.Zdvizka_HornaPoloha AND P3_ZdvizkaZaLeakTestB.IN.TlmicPaletky_ZASUNUTY THEN
				P3_ZdvizkaZaLeakTestB.OUT.TlmicPaletky_VYSUN:= FALSE;
				P3_ZdvizkaZaLeakTestB.OUT.TlmicPaletky_ZASUN:= FALSE;
				SC_P3_ZdvizkaZaLeakTestA.ResetStep:= TRUE;
				SC_P3_ZdvizkaZaLeakTestA.Step:= 123;
			END_IF

		123:
			SC_P3_ZdvizkaZaLeakTestA.StepName:='123 - Automaticky Rezim - cakam na ukoncenie vyvazania na Trat B';
			SC_P3_ZdvizkaZaLeakTestA.IdleTime.PT:= T#500ms;
			SC_P3_ZdvizkaZaLeakTestA.AlarmTime.PT:= T#5s;

			SC_P3_ZdvizkaZaLeakTestA.IdleTime.IN:= P3_ZdvizkaZaLeakTestB.IN.PritomnostPaletky AND P3_ZdvizkaZaLeakTestB.IN.PoziciaPaletky_OK;

			IF NOT SC_P3_ZdvizkaZaLeakTestA.Switch1 THEN
				P3_Dopravniky.OUT.PriecnyDopravnik2_VZAD:= FALSE;
				P3_Dopravniky.OUT.PriecnyDopravnik2_VPRED:= TRUE;
				SC_P3_ZdvizkaZaLeakTestA.Switch1:= TRUE;
			END_IF

			IF SC_P3_ZdvizkaZaLeakTestA.IdleTime.Q THEN
				P3_Dopravniky.OUT.PriecnyDopravnik2_VZAD:= FALSE;
				P3_Dopravniky.OUT.PriecnyDopravnik2_VPRED:= FALSE;
				SC_P3_ZdvizkaZaLeakTestA.ResetStep:= TRUE;
				SC_P3_ZdvizkaZaLeakTestA.Step:= 125;
			END_IF

		125:
			SC_P3_ZdvizkaZaLeakTestA.StepName:='123 - Automaticky Rezim - cakam na presun zdviziek do strednej polohy';
			SC_P3_ZdvizkaZaLeakTestA.IdleTime.PT:= T#1s;
			SC_P3_ZdvizkaZaLeakTestA.AlarmTime.PT:= T#5s;

			IF NOT SC_P3_ZdvizkaZaLeakTestA.Switch1 AND SC_OvlZdvizky.Step = 1 THEN
				Zdvizku_VYSTRED:= TRUE;
				P3_ZdvizkaZaLeakTestB.OUT.Zdvizku_ZASUN:= FALSE;
				P3_ZdvizkaZaLeakTestB.OUT.Zdvizku_VYSUN:= FALSE;
				SC_P3_ZdvizkaZaLeakTestA.Switch1:= TRUE;
			END_IF

			IF P3_ZdvizkaZaLeakTestA.IN.Zdvizka_StrednaPoloha AND P3_ZdvizkaZaLeakTestB.IN.Zdvizka_StrednaPoloha THEN
				P3_ZdvizkaZaLeakTestA.STAV.PrebiehaVyvezeniePaletkyNaTratB:= FALSE;
				SC_P3_ZdvizkaZaLeakTestA.ResetStep:= TRUE;
				SC_P3_ZdvizkaZaLeakTestA.Step:= 130;
			END_IF

			//Vysunutie tlmenia paletky//

		130:
			SC_P3_ZdvizkaZaLeakTestA.StepName:='130 - Automaticky Rezim - vysunutie tlamena paletky';
			SC_P3_ZdvizkaZaLeakTestA.IdleTime.PT:= T#1s;
			SC_P3_ZdvizkaZaLeakTestA.AlarmTime.PT:= T#5s;

			SC_P3_ZdvizkaZaLeakTestA.IdleTime.IN:= NOT P3_ZdvizkaZaLeakTestA.IN.TlmicPaletky_ZASUNUTY;

			IF NOT SC_P3_ZdvizkaZaLeakTestA.Switch1 THEN
				P3_ZdvizkaZaLeakTestA.OUT.TlmicPaletky_ZASUN:= FALSE;
				P3_ZdvizkaZaLeakTestA.OUT.TlmicPaletky_VYSUN:= TRUE;
				SC_P3_ZdvizkaZaLeakTestA.Switch1:= TRUE;
			END_IF

			IF SC_P3_ZdvizkaZaLeakTestA.IdleTime.Q THEN
				P3_ZdvizkaZaLeakTestA.OUT.TlmicPaletky_ZASUN:= FALSE;
				P3_ZdvizkaZaLeakTestA.OUT.TlmicPaletky_VYSUN:= FALSE;
				SC_P3_ZdvizkaZaLeakTestA.ResetStep:= TRUE;
				SC_P3_ZdvizkaZaLeakTestA.Step:= 100;
			END_IF

			//*******************************************************Manuálny režim*******************************************************************************//
		700:
			SC_P3_ZdvizkaZaLeakTestA.StepName:='700 - Manualny Rezim';
			SC_P3_ZdvizkaZaLeakTestA.IdleTime.PT:= T#8s;
			SC_P3_ZdvizkaZaLeakTestA.AlarmTime.PT:= T#5s;

	END_CASE

END_PROGRAM

PROGRAM _EXIT
	(* Insert code here *)

END_PROGRAM
```

#### Variables.var - Local variables
```iecst
VAR
	SC_OvlZdvizky : SequenceControlTyp;
	Zdvizku_VYSUN : BOOL;
	Zdvizku_ZASUN : BOOL;
	Zdvizku_VYSTRED : BOOL := FALSE;
END_VAR
```

#### OvlZdvizky.st
```iecst
ACTION OvlZdvizky:

	//Volanie funkcie SequenceControl//
	SequenceControl(SC:= SC_OvlZdvizky);

	CASE SC_OvlZdvizky.Step OF

		0:
			SC_OvlZdvizky.StepName:= '0 - Nulovanie';
			Zdvizku_VYSUN:= FALSE;
			Zdvizku_ZASUN:= FALSE;
			Zdvizku_VYSTRED:= FALSE;

			IF SC_P3_ZdvizkaZaLeakTestA.Step <> 0 THEN
				SC_OvlZdvizky.ResetStep:= TRUE;
				SC_OvlZdvizky.Step:= 1;
			END_IF

		1:
			SC_OvlZdvizky.StepName:= '1 - Rozhodnutie o cinnosti';
			IF Zdvizku_VYSUN THEN
				SC_OvlZdvizky.Step:= 10;
			ELSIF Zdvizku_ZASUN THEN
				SC_OvlZdvizky.Step:= 20;
			ELSIF Zdvizku_VYSTRED THEN
				SC_OvlZdvizky.Step:= 30;
			END_IF

		10:
			SC_OvlZdvizky.StepName:= '10 - Vysunutie zdvizky hore';
			SC_OvlZdvizky.IdleTime.PT:= T#3s;
			SC_OvlZdvizky.AlarmTime.PT:= T#6s;

			IF P3_ZdvizkaZaLeakTestA.Automat THEN
				SC_OvlZdvizky.AlarmTime.IN:= TRUE;
			ELSE
				SC_OvlZdvizky.IdleTime.IN:= TRUE;
			END_IF

			IF NOT SC_OvlZdvizky.Switch1 THEN
				P3_ZdvizkaZaLeakTestA.OUT.Zdvizku_ZASUN:= FALSE;
				P3_ZdvizkaZaLeakTestA.OUT.Zdvizku_VYSUN:= TRUE;
				SC_OvlZdvizky.Switch1:= TRUE;
			END_IF

			IF P3_ZdvizkaZaLeakTestA.IN.Zdvizka_HornaPoloha OR SC_OvlZdvizky.IdleTime.Q THEN
				SC_OvlZdvizky.ResetStep:= TRUE;
				SC_OvlZdvizky.Step:= 0;
			ELSIF SC_OvlZdvizky.AlarmTime.Q THEN
				P34_Alarmy[374]:= TRUE;
				P3_Pracovisko.STAV.Porucha_ST7:= TRUE;
			END_IF

		20:
			SC_OvlZdvizky.StepName:= '20 - Zasunutie zdvizky dole';
			SC_OvlZdvizky.IdleTime.PT:= T#3s;
			SC_OvlZdvizky.AlarmTime.PT:= T#6s;

			IF P3_ZdvizkaZaLeakTestA.Automat THEN
				SC_OvlZdvizky.AlarmTime.IN:= TRUE;
			ELSE
				SC_OvlZdvizky.IdleTime.IN:= TRUE;
			END_IF

			IF NOT SC_OvlZdvizky.Switch1 THEN
				P3_ZdvizkaZaLeakTestA.OUT.Zdvizku_VYSUN:= FALSE;
				P3_ZdvizkaZaLeakTestA.OUT.Zdvizku_ZASUN:= TRUE;
				SC_OvlZdvizky.Switch1:= TRUE;
			END_IF

			IF P3_ZdvizkaZaLeakTestA.IN.Zdvizka_SpodnaPoloha OR SC_OvlZdvizky.IdleTime.Q THEN
				SC_OvlZdvizky.ResetStep:= TRUE;
				SC_OvlZdvizky.Step:= 0;
			ELSIF SC_OvlZdvizky.AlarmTime.Q THEN
				P34_Alarmy[375]:= TRUE;
				P3_Pracovisko.STAV.Porucha_ST7:= TRUE;
			END_IF

		30:
			SC_OvlZdvizky.StepName:= '30 - Presun zdvizky do strednej polohy';
			SC_OvlZdvizky.IdleTime.PT:= T#3s;
			SC_OvlZdvizky.AlarmTime.PT:= T#6s;

			IF P3_ZdvizkaZaLeakTestA.Automat THEN
				SC_OvlZdvizky.AlarmTime.IN:= TRUE;
			ELSE
				SC_OvlZdvizky.IdleTime.IN:= TRUE;
			END_IF

			IF NOT SC_OvlZdvizky.Switch1 THEN
				P3_ZdvizkaZaLeakTestA.OUT.Zdvizku_VYSUN:= FALSE;
				P3_ZdvizkaZaLeakTestA.OUT.Zdvizku_ZASUN:= FALSE;
				SC_OvlZdvizky.Switch1:= TRUE;
			END_IF

			IF P3_ZdvizkaZaLeakTestA.IN.Zdvizka_StrednaPoloha OR SC_OvlZdvizky.IdleTime.Q THEN
				SC_OvlZdvizky.ResetStep:= TRUE;
				SC_OvlZdvizky.Step:= 0;
			ELSIF SC_OvlZdvizky.AlarmTime.Q THEN
				P34_Alarmy[376]:= TRUE;
				P3_Pracovisko.STAV.Porucha_ST7:= TRUE;
			END_IF

	END_CASE

END_ACTION
```

### Program Logical/Program/Pracovisko_3/P3_ZdvizkaZaLeakTestB (IEC)

#### Main.st - Init, cyclic, exit code
```iecst
PROGRAM _INIT
	(* Insert code here *)

END_PROGRAM

PROGRAM _CYCLIC

	//Volanie funkcie SequenceControl//
	SequenceControl(SC:= SC_P3_ZdvizkaZaLeakTestB);

	//Volanie podprogramov//
	OvlZdvizky;

	//Reset sekcie //
	IF P3_ZdvizkaZaLeakTestB.Reset THEN
		SC_P3_ZdvizkaZaLeakTestB.Step:= 0;
		P3_ZdvizkaZaLeakTestB.Reset:= FALSE;
	ELSIF NOT Safety.STAV.Linka_ZonaCS_AKTIVNA THEN
		SC_P3_ZdvizkaZaLeakTestB.Step:= 0;
	END_IF

	CASE SC_P3_ZdvizkaZaLeakTestB.Step OF

		0:
			SC_P3_ZdvizkaZaLeakTestB.StepName:='0 - Nulovanie';
			SC_OvlZdvizky.Step:= 0;
			P3_ZdvizkaZaLeakTestB.Automat:= FALSE;
			P3_ZdvizkaZaLeakTestB.KoniecCyklu:= FALSE;
			P3_ZdvizkaZaLeakTestB.Manual:= FALSE;
			P3_ZdvizkaZaLeakTestB.STAV.PoINIT:= FALSE;
			P3_ZdvizkaZaLeakTestB.OUT.TlmicPaletky_VYSUN:= FALSE;
			P3_ZdvizkaZaLeakTestB.OUT.TlmicPaletky_ZASUN:= FALSE;
			P3_Dopravniky.OUT.PriecnyDopravnik2_VPRED:= FALSE;
			P3_Dopravniky.OUT.PriecnyDopravnik2_VZAD:= FALSE;
			P3_ZdvizkaZaLeakTestB.STAV.PrebiehaVyvezeniePaletkyNaTratA:= FALSE;
			P3_ZdvizkaZaLeakTestB.STAV.PrebiehaVyvezeniePaletkyNaTratB:= FALSE;
			P3_LeakageTestB.STAV.PrebiehaVyvezeniePaletky:= FALSE;

			IF Safety.STAV.Linka_ZonaCS_AKTIVNA AND
				Safety.STAV.P3_ZonaBunky_AKTIVNA AND
				P3_Pracovisko.STAV.HardwareBunky_OK AND
				NOT P3_Pracovisko.STAV.Porucha_ST1 AND
				NOT P3_Pracovisko.STAV.Porucha_ST2 AND
				NOT P3_Pracovisko.STAV.Porucha_ST3 AND
				NOT P3_Pracovisko.STAV.Porucha_ST4 AND
				NOT P3_Pracovisko.STAV.Porucha_ST5 AND
				NOT P3_Pracovisko.STAV.Porucha_ST6 AND
				NOT P3_Pracovisko.STAV.Porucha_ST7 AND
				NOT P3_Pracovisko.STAV.Porucha_ST8 THEN
				SC_P3_ZdvizkaZaLeakTestB.ResetStep:= TRUE;
				SC_P3_ZdvizkaZaLeakTestB.Step:= 1;
			END_IF

		1:
			SC_P3_ZdvizkaZaLeakTestB.StepName:='1 - Cakam na spustenie vyroby';
			P3_ZdvizkaZaLeakTestB.KoniecCyklu:= FALSE;
			IF P3_ZdvizkaZaLeakTestB.Automat THEN
				SC_P3_ZdvizkaZaLeakTestB.Step:= 2;
			ELSIF P3_ZdvizkaZaLeakTestB.Manual THEN
				SC_P3_ZdvizkaZaLeakTestB.Step:= 700;
			END_IF

			//********************************************************Inicializácia****************************************************************************//

		2:
			SC_P3_ZdvizkaZaLeakTestB.StepName:='2 - Inicializacia - cakam na spustenie inicializacie';
			SC_P3_ZdvizkaZaLeakTestB.IdleTime.PT:= T#500ms;
			SC_P3_ZdvizkaZaLeakTestB.AlarmTime.PT:= T#5s;

			IF P3_Dopravniky.STAV.PoINIT THEN
				SC_P3_ZdvizkaZaLeakTestB.ResetStep:= TRUE;
				SC_P3_ZdvizkaZaLeakTestB.Step:= 5;
			END_IF

		5:
			SC_P3_ZdvizkaZaLeakTestB.StepName:='5 - Inicializacia - kontrola pozicie zdvizky';
			SC_P3_ZdvizkaZaLeakTestB.IdleTime.PT:= T#500ms;
			SC_P3_ZdvizkaZaLeakTestB.AlarmTime.PT:= T#5s;

			IF P3_ZdvizkaZaLeakTestB.IN.Zdvizka_StrednaPoloha AND P3_ZdvizkaZaLeakTestB.IN.PritomnostPaletky THEN
				P3_ZdvizkaZaLeakTestB.STAV.PoINIT:= TRUE;
				SC_P3_ZdvizkaZaLeakTestB.ResetStep:= TRUE;
				SC_P3_ZdvizkaZaLeakTestB.Step:= 100;
			ELSE
				SC_P3_ZdvizkaZaLeakTestB.ResetStep:= TRUE;
				SC_P3_ZdvizkaZaLeakTestB.Step:= 8;
			END_IF

		8:
			SC_P3_ZdvizkaZaLeakTestB.StepName:='8 - Inicializacia - presun zdvizky do hornej polohy';
			SC_P3_ZdvizkaZaLeakTestB.IdleTime.PT:= T#500ms;
			SC_P3_ZdvizkaZaLeakTestB.AlarmTime.PT:= T#5s;

			IF NOT SC_P3_ZdvizkaZaLeakTestB.Switch1 AND SC_OvlZdvizky.Step = 1 THEN
				Zdvizku_VYSUN:= TRUE;
				P3_ZdvizkaZaLeakTestB.OUT.TlmicPaletky_VYSUN:= FALSE;
				P3_ZdvizkaZaLeakTestB.OUT.TlmicPaletky_ZASUN:= TRUE;
				SC_P3_ZdvizkaZaLeakTestB.Switch1:= TRUE;
			END_IF

			IF P3_ZdvizkaZaLeakTestB.IN.Zdvizka_HornaPoloha AND P3_ZdvizkaZaLeakTestB.IN.TlmicPaletky_ZASUNUTY THEN
				SC_P3_ZdvizkaZaLeakTestB.ResetStep:= TRUE;
				SC_P3_ZdvizkaZaLeakTestB.Step:= 10;
			END_IF

		10:
			SC_P3_ZdvizkaZaLeakTestB.StepName:='10 - Inicializacia - kontrola pritomnosti paletky na zdvizke za Leakage Testom A';
			SC_P3_ZdvizkaZaLeakTestB.IdleTime.PT:= T#500ms;
			SC_P3_ZdvizkaZaLeakTestB.AlarmTime.PT:= T#5s;

			IF NOT P3_ZdvizkaZaLeakTestA.IN.PritomnostPaletky THEN
				P3_ZdvizkaZaLeakTestA.OUT.Zdvizku_ZASUN:= FALSE;
				P3_ZdvizkaZaLeakTestA.OUT.Zdvizku_VYSUN:= TRUE;
				SC_P3_ZdvizkaZaLeakTestB.ResetStep:= TRUE;
				SC_P3_ZdvizkaZaLeakTestB.Step:= 11;
			ELSE
				SC_P3_ZdvizkaZaLeakTestB.ResetStep:= TRUE;
				SC_P3_ZdvizkaZaLeakTestB.Step:= 13;
			END_IF

		11:
			SC_P3_ZdvizkaZaLeakTestB.StepName:='11 - Inicializacia - cakam na zodvihnutie zdvizky za Leakage Testom A';
			SC_P3_ZdvizkaZaLeakTestB.IdleTime.PT:= T#500ms;
			SC_P3_ZdvizkaZaLeakTestB.AlarmTime.PT:= T#5s;

			IF P3_ZdvizkaZaLeakTestA.IN.Zdvizka_HornaPoloha THEN
				SC_P3_ZdvizkaZaLeakTestB.ResetStep:= TRUE;
				SC_P3_ZdvizkaZaLeakTestB.Step:= 13;
			END_IF

		13:
			SC_P3_ZdvizkaZaLeakTestB.StepName:='13 - Inicializacia - spustenie priecneho dopravnika';
			SC_P3_ZdvizkaZaLeakTestB.IdleTime.PT:= T#500ms;
			SC_P3_ZdvizkaZaLeakTestB.AlarmTime.PT:= T#7s;

			SC_P3_ZdvizkaZaLeakTestB.IdleTime.IN:= P3_ZdvizkaZaLeakTestB.IN.PritomnostPaletky AND P3_ZdvizkaZaLeakTestB.IN.PoziciaPaletky_OK;

			IF NOT SC_P3_ZdvizkaZaLeakTestB.Switch1 THEN
				P3_Dopravniky.OUT.PriecnyDopravnik2_VZAD:= FALSE;
				P3_Dopravniky.OUT.PriecnyDopravnik2_VPRED:= TRUE;
				SC_P3_ZdvizkaZaLeakTestB.AlarmTime.IN:= TRUE;
				SC_P3_ZdvizkaZaLeakTestB.Switch1:= TRUE;
			END_IF

			IF SC_P3_ZdvizkaZaLeakTestB.IdleTime.Q THEN
				P3_Dopravniky.OUT.PriecnyDopravnik2_VZAD:= FALSE;
				P3_Dopravniky.OUT.PriecnyDopravnik2_VPRED:= FALSE;
				SC_P3_ZdvizkaZaLeakTestB.ResetStep:= TRUE;
				SC_P3_ZdvizkaZaLeakTestB.Step:= 15;
			ELSIF SC_P3_ZdvizkaZaLeakTestB.AlarmTime.Q THEN
				P3_Dopravniky.OUT.PriecnyDopravnik2_VZAD:= FALSE;
				P3_Dopravniky.OUT.PriecnyDopravnik2_VPRED:= FALSE;
				SC_P3_ZdvizkaZaLeakTestB.ResetStep:= TRUE;
				SC_P3_ZdvizkaZaLeakTestB.Step:= 15;
			END_IF

		15:
			SC_P3_ZdvizkaZaLeakTestB.StepName:='15 - Inicializacia - presun zdvizky do strednej polohy';
			SC_P3_ZdvizkaZaLeakTestB.IdleTime.PT:= T#500ms;
			SC_P3_ZdvizkaZaLeakTestB.AlarmTime.PT:= T#5s;

			IF NOT SC_P3_ZdvizkaZaLeakTestB.Switch1 AND SC_OvlZdvizky.Step = 1 THEN
				Zdvizku_VYSTRED:= TRUE;
				P3_ZdvizkaZaLeakTestA.OUT.Zdvizku_ZASUN:= FALSE;
				P3_ZdvizkaZaLeakTestA.OUT.Zdvizku_VYSUN:= FALSE;
				SC_P3_ZdvizkaZaLeakTestB.Switch1:= TRUE;
			END_IF

			IF P3_ZdvizkaZaLeakTestB.IN.Zdvizka_StrednaPoloha AND P3_ZdvizkaZaLeakTestA.IN.Zdvizka_StrednaPoloha THEN
				IF P3_ZdvizkaZaLeakTestB.IN.PritomnostPaletky THEN
					P3_ZdvizkaZaLeakTestB.STAV.PoINIT:= TRUE;
					SC_P3_ZdvizkaZaLeakTestB.ResetStep:= TRUE;
					SC_P3_ZdvizkaZaLeakTestB.Step:= 100;
				ELSE
					SC_P3_ZdvizkaZaLeakTestB.ResetStep:= TRUE;
					SC_P3_ZdvizkaZaLeakTestB.Step:= 18;
				END_IF
			END_IF

		18:
			SC_P3_ZdvizkaZaLeakTestB.StepName:='18 - Inicializacia - vysunutie tlmica paletky';
			SC_P3_ZdvizkaZaLeakTestB.IdleTime.PT:= T#500ms;
			SC_P3_ZdvizkaZaLeakTestB.AlarmTime.PT:= T#5s;

			IF NOT SC_P3_ZdvizkaZaLeakTestB.Switch1 THEN
				P3_ZdvizkaZaLeakTestB.OUT.TlmicPaletky_ZASUN:= FALSE;
				P3_ZdvizkaZaLeakTestB.OUT.TlmicPaletky_VYSUN:= TRUE;
				SC_P3_ZdvizkaZaLeakTestB.IdleTime.IN:= TRUE;
				SC_P3_ZdvizkaZaLeakTestB.Switch1:= TRUE;
			END_IF

			IF SC_P3_ZdvizkaZaLeakTestB.IdleTime.Q THEN
				P3_ZdvizkaZaLeakTestB.OUT.TlmicPaletky_ZASUN:= FALSE;
				P3_ZdvizkaZaLeakTestB.OUT.TlmicPaletky_VYSUN:= FALSE;
				P3_ZdvizkaZaLeakTestB.STAV.PoINIT:= TRUE;
				SC_P3_ZdvizkaZaLeakTestB.ResetStep:= TRUE;
				SC_P3_ZdvizkaZaLeakTestB.Step:= 100;
			END_IF

			//********************************************************Automatický režim****************************************************************************//
		100:
			SC_P3_ZdvizkaZaLeakTestB.StepName:='100 - Automaticky Rezim - cakam na príchod paletky na zdvizku';
			SC_P3_ZdvizkaZaLeakTestB.IdleTime.PT:= T#200ms;
			SC_P3_ZdvizkaZaLeakTestB.AlarmTime.PT:= T#5s;

			SC_P3_ZdvizkaZaLeakTestB.IdleTime.IN:= P3_ZdvizkaZaLeakTestB.IN.PritomnostPaletky AND P3_ZdvizkaZaLeakTestB.IN.TlmicPaletky_ZASUNUTY AND P3_ZdvizkaZaLeakTestB.IN.PoziciaPaletky_OK AND P3_ZdvizkaZaLeakTestB.IN.Zdvizka_StrednaPoloha;

			IF P3_ZdvizkaZaLeakTestB.IN.PritomnostPaletky AND P3_ZdvizkaZaLeakTestB.IN.Zdvizka_StrednaPoloha THEN
				P3_LeakageTestB.STAV.PrebiehaVyvezeniePaletky:= FALSE;
				P3_ZdvizkaZaLeakTestA.STAV.PrebiehaVyvezeniePaletkyNaTratB:= FALSE;
			END_IF

			IF P3_ZdvizkaZaLeakTestB.KoniecCyklu AND NOT P3_LeakageTestB.Automat THEN
				SC_P3_ZdvizkaZaLeakTestB.ResetStep:= TRUE;
				SC_P3_ZdvizkaZaLeakTestB.Step:= 0;
			ELSIF SC_P3_ZdvizkaZaLeakTestB.IdleTime.Q THEN
				SC_P3_ZdvizkaZaLeakTestB.ResetStep:= TRUE;
				SC_P3_ZdvizkaZaLeakTestB.Step:= 101;
			END_IF

		101:
			SC_P3_ZdvizkaZaLeakTestB.StepName:='101 - Automaticky Rezim - rozhodnutie o smere vyvazania';
			SC_P3_ZdvizkaZaLeakTestB.IdleTime.PT:= T#200ms;
			SC_P3_ZdvizkaZaLeakTestB.AlarmTime.PT:= T#5s;

			IF P3_ZdvizkaZaLeakTestB.KoniecCyklu AND NOT P3_LeakageTestB.Automat THEN
				SC_P3_ZdvizkaZaLeakTestB.ResetStep:= TRUE;
				SC_P3_ZdvizkaZaLeakTestB.Step:= 0;
			ELSIF P4_FunkcnyTestB.STAV.Tester_ON AND  //Vyvážanie na trať B
				NOT P4_FunkcnyTestB.RFID_hlava.PritomnostPaletky AND
				SC_P4_FunkcnyTestB.Step = 100 AND
				NOT P3_ZdvizkaZaLeakTestB.STAV.PrebiehaVyvezeniePaletkyNaTratB AND
				NOT P3_ZdvizkaZaLeakTestA.STAV.PrebiehaVyvezeniePaletkyNaTratB THEN
				SC_P3_ZdvizkaZaLeakTestB.ResetStep:= TRUE;
				SC_P3_ZdvizkaZaLeakTestB.Step:= 110;
			ELSIF NOT P4_FunkcnyTestB.STAV.Tester_ON AND  //Vyvážanie na trať A//
				P4_FunkcnyTestA.STAV.Tester_ON AND
				NOT P3_ZdvizkaZaLeakTestA.IN.PritomnostPaletky AND
				SC_P3_ZdvizkaZaLeakTestA.Step = 100 AND
				NOT P3_ZdvizkaZaLeakTestA.STAV.PrebiehaVyvezeniePaletkyNaTratB AND
				NOT P3_LeakageTestA.STAV.PrebiehaVyvezeniePaletky AND
				SC_P3_LeakageTestA.Step < 560  THEN
				SC_P3_ZdvizkaZaLeakTestB.ResetStep:= TRUE;
				SC_P3_ZdvizkaZaLeakTestB.Step:= 120;
			ELSIF NOT P3_ZdvizkaZaLeakTestB.IN.PritomnostPaletky THEN
				SC_P3_ZdvizkaZaLeakTestB.ResetStep:= TRUE;
				SC_P3_ZdvizkaZaLeakTestB.Step:= 100;
			END_IF

			//Vyvážanie na trať B//
		110:
			SC_P3_ZdvizkaZaLeakTestB.StepName:='110 - Automaticky Rezim - presun zdvizky do spodnej polohy';
			SC_P3_ZdvizkaZaLeakTestB.IdleTime.PT:= T#200ms;
			SC_P3_ZdvizkaZaLeakTestB.AlarmTime.PT:= T#5s;

			IF NOT SC_P3_ZdvizkaZaLeakTestB.Switch1 AND SC_OvlZdvizky.Step = 1 THEN
				Zdvizku_ZASUN:= TRUE;
				P3_ZdvizkaZaLeakTestB.STAV.PrebiehaVyvezeniePaletkyNaTratB:= TRUE;
				SC_P3_ZdvizkaZaLeakTestB.Switch1:= TRUE;
			END_IF

			IF P3_ZdvizkaZaLeakTestB.IN.Zdvizka_SpodnaPoloha THEN
				SC_P3_ZdvizkaZaLeakTestB.ResetStep:= TRUE;
				SC_P3_ZdvizkaZaLeakTestB.Step:= 113;
			END_IF

		113:
			SC_P3_ZdvizkaZaLeakTestB.StepName:='113 - Automaticky Rezim - cakam na ukoncenie vyvazania na Trat B';
			SC_P3_ZdvizkaZaLeakTestB.IdleTime.PT:= T#500ms;
			SC_P3_ZdvizkaZaLeakTestB.AlarmTime.PT:= T#5s;

			SC_P3_ZdvizkaZaLeakTestB.IdleTime.IN:= NOT P3_ZdvizkaZaLeakTestB.IN.PritomnostPaletky;

			IF SC_P3_ZdvizkaZaLeakTestB.IdleTime.Q AND NOT SC_P3_ZdvizkaZaLeakTestB.Switch1 AND SC_OvlZdvizky.Step = 1 THEN
				Zdvizku_VYSTRED:= TRUE;
				SC_P3_ZdvizkaZaLeakTestB.Switch1:= TRUE;
			END_IF

			IF P3_ZdvizkaZaLeakTestB.IN.Zdvizka_StrednaPoloha THEN
				SC_P3_ZdvizkaZaLeakTestB.ResetStep:= TRUE;
				SC_P3_ZdvizkaZaLeakTestB.Step:= 130;
			END_IF

			//Vyvážanie na trať A//
		120:
			SC_P3_ZdvizkaZaLeakTestB.StepName:='120 - Automaticky Rezim - presun zdviziek do hornej polohy';
			SC_P3_ZdvizkaZaLeakTestB.IdleTime.PT:= T#200ms;
			SC_P3_ZdvizkaZaLeakTestB.AlarmTime.PT:= T#5s;

			IF NOT SC_P3_ZdvizkaZaLeakTestB.Switch1 AND SC_OvlZdvizky.Step = 1 THEN
				Zdvizku_VYSUN:= TRUE;
				P3_ZdvizkaZaLeakTestA.OUT.Zdvizku_ZASUN:= FALSE;
				P3_ZdvizkaZaLeakTestA.OUT.Zdvizku_VYSUN:= TRUE;
				P3_ZdvizkaZaLeakTestA.OUT.TlmicPaletky_VYSUN:= FALSE;
				P3_ZdvizkaZaLeakTestA.OUT.TlmicPaletky_ZASUN:= TRUE;
				P3_ZdvizkaZaLeakTestB.STAV.PrebiehaVyvezeniePaletkyNaTratA:= TRUE;
				SC_P3_ZdvizkaZaLeakTestB.Switch1:= TRUE;
			END_IF

			IF P3_ZdvizkaZaLeakTestA.IN.Zdvizka_HornaPoloha AND P3_ZdvizkaZaLeakTestB.IN.Zdvizka_HornaPoloha AND P3_ZdvizkaZaLeakTestA.IN.TlmicPaletky_ZASUNUTY THEN
				P3_ZdvizkaZaLeakTestA.OUT.TlmicPaletky_VYSUN:= FALSE;
				P3_ZdvizkaZaLeakTestA.OUT.TlmicPaletky_ZASUN:= FALSE;
				SC_P3_ZdvizkaZaLeakTestB.ResetStep:= TRUE;
				SC_P3_ZdvizkaZaLeakTestB.Step:= 123;
			END_IF

		123:
			SC_P3_ZdvizkaZaLeakTestB.StepName:='123 - Automaticky Rezim - cakam na ukoncenie vyvazania na Trat A';
			SC_P3_ZdvizkaZaLeakTestB.IdleTime.PT:= T#500ms;
			SC_P3_ZdvizkaZaLeakTestB.AlarmTime.PT:= T#5s;

			SC_P3_ZdvizkaZaLeakTestB.IdleTime.IN:= P3_ZdvizkaZaLeakTestA.IN.PritomnostPaletky;

			IF NOT SC_P3_ZdvizkaZaLeakTestB.Switch1 THEN
				P3_Dopravniky.OUT.PriecnyDopravnik2_VPRED:= FALSE;
				P3_Dopravniky.OUT.PriecnyDopravnik2_VZAD:= TRUE;
				SC_P3_ZdvizkaZaLeakTestB.Switch1:= TRUE;
			END_IF

			IF SC_P3_ZdvizkaZaLeakTestB.IdleTime.Q THEN
				P3_Dopravniky.OUT.PriecnyDopravnik2_VZAD:= FALSE;
				P3_Dopravniky.OUT.PriecnyDopravnik2_VPRED:= FALSE;
				SC_P3_ZdvizkaZaLeakTestB.ResetStep:= TRUE;
				SC_P3_ZdvizkaZaLeakTestB.Step:= 125;
			END_IF

		125:
			SC_P3_ZdvizkaZaLeakTestB.StepName:='123 - Automaticky Rezim - cakam na presun zdviziek do strednej polohy';
			SC_P3_ZdvizkaZaLeakTestB.IdleTime.PT:= T#1s;
			SC_P3_ZdvizkaZaLeakTestB.AlarmTime.PT:= T#5s;

			IF NOT SC_P3_ZdvizkaZaLeakTestB.Switch1 AND SC_OvlZdvizky.Step = 1 THEN
				Zdvizku_VYSTRED:= TRUE;
				P3_ZdvizkaZaLeakTestA.OUT.Zdvizku_ZASUN:= FALSE;
				P3_ZdvizkaZaLeakTestA.OUT.Zdvizku_VYSUN:= FALSE;
				SC_P3_ZdvizkaZaLeakTestB.Switch1:= TRUE;
			END_IF

			IF P3_ZdvizkaZaLeakTestA.IN.Zdvizka_StrednaPoloha AND P3_ZdvizkaZaLeakTestB.IN.Zdvizka_StrednaPoloha THEN
				P3_ZdvizkaZaLeakTestB.STAV.PrebiehaVyvezeniePaletkyNaTratA:= FALSE;
				SC_P3_ZdvizkaZaLeakTestB.ResetStep:= TRUE;
				SC_P3_ZdvizkaZaLeakTestB.Step:= 130;
			END_IF

		//Vysunutie tlmenia paletky//

		130:
			SC_P3_ZdvizkaZaLeakTestB.StepName:='130 - Automaticky Rezim - vysunutie tlamena paletky';
			SC_P3_ZdvizkaZaLeakTestB.IdleTime.PT:= T#1s;
			SC_P3_ZdvizkaZaLeakTestB.AlarmTime.PT:= T#5s;

			SC_P3_ZdvizkaZaLeakTestB.IdleTime.IN:= NOT P3_ZdvizkaZaLeakTestB.IN.TlmicPaletky_ZASUNUTY;

			IF NOT SC_P3_ZdvizkaZaLeakTestB.Switch1 THEN
				P3_ZdvizkaZaLeakTestB.OUT.TlmicPaletky_ZASUN:= FALSE;
				P3_ZdvizkaZaLeakTestB.OUT.TlmicPaletky_VYSUN:= TRUE;
				SC_P3_ZdvizkaZaLeakTestB.Switch1:= TRUE;
			END_IF

			IF SC_P3_ZdvizkaZaLeakTestB.IdleTime.Q THEN
				P3_ZdvizkaZaLeakTestB.OUT.TlmicPaletky_ZASUN:= FALSE;
				P3_ZdvizkaZaLeakTestB.OUT.TlmicPaletky_VYSUN:= FALSE;
				SC_P3_ZdvizkaZaLeakTestB.ResetStep:= TRUE;
				SC_P3_ZdvizkaZaLeakTestB.Step:= 100;
			END_IF

			//*******************************************************Manuálny režim*******************************************************************************//
		700:
			SC_P3_ZdvizkaZaLeakTestB.StepName:='700 - Manualny Rezim';
			SC_P3_ZdvizkaZaLeakTestB.IdleTime.PT:= T#8s;
			SC_P3_ZdvizkaZaLeakTestB.AlarmTime.PT:= T#5s;

	END_CASE

END_PROGRAM

PROGRAM _EXIT
	(* Insert code here *)

END_PROGRAM
```

#### Variables.var - Local variables
```iecst
VAR
	SC_OvlZdvizky : SequenceControlTyp;
	Zdvizku_VYSUN : BOOL;
	Zdvizku_ZASUN : BOOL;
	Zdvizku_VYSTRED : BOOL := FALSE;
END_VAR
```

#### OvlZdvizky.st
```iecst
ACTION OvlZdvizky:

	//Volanie funkcie SequenceControl//
	SequenceControl(SC:= SC_OvlZdvizky);

	CASE SC_OvlZdvizky.Step OF

		0:
			SC_OvlZdvizky.StepName:= '0 - Nulovanie';
			Zdvizku_VYSUN:= FALSE;
			Zdvizku_ZASUN:= FALSE;
			Zdvizku_VYSTRED:= FALSE;

			IF SC_P3_ZdvizkaZaLeakTestB.Step <> 0 THEN
				SC_OvlZdvizky.ResetStep:= TRUE;
				SC_OvlZdvizky.Step:= 1;
			END_IF

		1:
			SC_OvlZdvizky.StepName:= '1 - Rozhodnutie o cinnosti';
			IF Zdvizku_VYSUN THEN
				SC_OvlZdvizky.Step:= 10;
			ELSIF Zdvizku_ZASUN THEN
				SC_OvlZdvizky.Step:= 20;
			ELSIF Zdvizku_VYSTRED THEN
				SC_OvlZdvizky.Step:= 30;
			END_IF

		10:
			SC_OvlZdvizky.StepName:= '10 - Vysunutie zdvizky hore';
			SC_OvlZdvizky.IdleTime.PT:= T#3s;
			SC_OvlZdvizky.AlarmTime.PT:= T#6s;

			IF P3_ZdvizkaZaLeakTestB.Automat THEN
				SC_OvlZdvizky.AlarmTime.IN:= TRUE;
			ELSE
				SC_OvlZdvizky.IdleTime.IN:= TRUE;
			END_IF

			IF NOT SC_OvlZdvizky.Switch1 THEN
				P3_ZdvizkaZaLeakTestB.OUT.Zdvizku_ZASUN:= FALSE;
				P3_ZdvizkaZaLeakTestB.OUT.Zdvizku_VYSUN:= TRUE;
				SC_OvlZdvizky.Switch1:= TRUE;
			END_IF

			IF P3_ZdvizkaZaLeakTestB.IN.Zdvizka_HornaPoloha OR SC_OvlZdvizky.IdleTime.Q THEN
				SC_OvlZdvizky.ResetStep:= TRUE;
				SC_OvlZdvizky.Step:= 0;
			ELSIF SC_OvlZdvizky.AlarmTime.Q THEN
				P34_Alarmy[377]:= TRUE;
				P3_Pracovisko.STAV.Porucha_ST8:= TRUE;
			END_IF

		20:
			SC_OvlZdvizky.StepName:= '20 - Zasunutie zdvizky dole';
			SC_OvlZdvizky.IdleTime.PT:= T#3s;
			SC_OvlZdvizky.AlarmTime.PT:= T#6s;

			IF P3_ZdvizkaZaLeakTestB.Automat THEN
				SC_OvlZdvizky.AlarmTime.IN:= TRUE;
			ELSE
				SC_OvlZdvizky.IdleTime.IN:= TRUE;
			END_IF

			IF NOT SC_OvlZdvizky.Switch1 THEN
				P3_ZdvizkaZaLeakTestB.OUT.Zdvizku_VYSUN:= FALSE;
				P3_ZdvizkaZaLeakTestB.OUT.Zdvizku_ZASUN:= TRUE;
				SC_OvlZdvizky.Switch1:= TRUE;
			END_IF

			IF P3_ZdvizkaZaLeakTestB.IN.Zdvizka_SpodnaPoloha OR SC_OvlZdvizky.IdleTime.Q THEN
				SC_OvlZdvizky.ResetStep:= TRUE;
				SC_OvlZdvizky.Step:= 0;
			ELSIF SC_OvlZdvizky.AlarmTime.Q THEN
				P34_Alarmy[378]:= TRUE;
				P3_Pracovisko.STAV.Porucha_ST8:= TRUE;
			END_IF

		30:
			SC_OvlZdvizky.StepName:= '30 - Presun zdvizky do strednej polohy';
			SC_OvlZdvizky.IdleTime.PT:= T#3s;
			SC_OvlZdvizky.AlarmTime.PT:= T#6s;

			IF P3_ZdvizkaZaLeakTestB.Automat THEN
				SC_OvlZdvizky.AlarmTime.IN:= TRUE;
			ELSE
				SC_OvlZdvizky.IdleTime.IN:= TRUE;
			END_IF

			IF NOT SC_OvlZdvizky.Switch1 THEN
				P3_ZdvizkaZaLeakTestB.OUT.Zdvizku_VYSUN:= FALSE;
				P3_ZdvizkaZaLeakTestB.OUT.Zdvizku_ZASUN:= FALSE;
				SC_OvlZdvizky.Switch1:= TRUE;
			END_IF

			IF P3_ZdvizkaZaLeakTestB.IN.Zdvizka_StrednaPoloha OR SC_OvlZdvizky.IdleTime.Q THEN
				SC_OvlZdvizky.ResetStep:= TRUE;
				SC_OvlZdvizky.Step:= 0;
			ELSIF SC_OvlZdvizky.AlarmTime.Q THEN
				P34_Alarmy[379]:= TRUE;
				P3_Pracovisko.STAV.Porucha_ST8:= TRUE;
			END_IF

	END_CASE

END_ACTION
```

### Program Logical/Program/Pracovisko_3/P3_Mapping_IO (IEC)
